gfCNCPoint2[3628] = {X 472.8698, Y 18.3782, Z -2.1667, A 0.000, B 0.000, C 0.000 }
gfCNCPoint2[3629] = {X 473.2481, Y 16.7251, Z -2.1667, A 0.000, B 0.000, C 0.000 }
gfCNCPoint2[3630] = {X 473.7840, Y 15.2312, Z -2.1667, A 0.000, B 0.000, C 0.000 }
gfCNCPoint2[3631] = {X 474.5174, Y 13.8238, Z -2.1667, A 0.000, B 0.000, C 0.000 }
gfCNCPoint2[3632] = {X 475.4350, Y 12.5288, Z -2.1667, A 0.000, B 0.000, C 0.000 }
gfCNCPoint2[3633] = {X 476.5196, Y 11.3702, Z -2.1667, A 0.000, B 0.000, C 0.000 }
gfCNCPoint2[3634] = {X 477.7513, Y 10.3694, Z -2.1667, A 0.000, B 0.000, C 0.000 }
gfCNCPoint2[3635] = {X 479.1074, Y 9.5448, Z -2.1667, A 0.000, B 0.000, C 0.000 }
gfCNCPoint2[3636] = {X 480.5628, Y 8.9117, Z -2.1667, A 0.000, B 0.000, C 0.000 }
gfCNCPoint2[3637] = {X 482.0905, Y 8.4819, Z -2.1667, A 0.000, B 0.000, C 0.000 }
gfCNCPoint2[3638] = {X 484.1725, Y 8.1580, Z -2.1667, A 0.000, B 0.000, C 0.000 }
gfCNCPoint2[3639] = {X 486.2764, Y 8.0437, Z -2.1667, A 0.000, B 0.000, C 0.000 }
gfCNCPoint2[3640] = {X 486.9693, Y 8.0316, Z -2.1667, A 0.000, B 0.000, C 0.000 }
gfCNCPoint2[3641] = {X 492.3824, Y 8.0316, Z -2.1667, A 0.000, B 0.000, C 0.000 }
gfCNCPoint2[3642] = {X 492.3824, Y 4.0316, Z -2.1667, A 0.000, B 0.000, C 0.000 }
gfCNCPoint2[3643] = {X 492.3824, Y 8.1116, Z -2.1667, A 0.000, B 0.000, C 0.000 }
gfCNCPoint2[3644] = {X 502.2056, Y 8.1116, Z -2.1667, A 0.000, B 0.000, C 0.000 }
gfCNCPoint2[3645] = {X 502.7355, Y 8.1157, Z -2.1667, A 0.000, B 0.000, C 0.000 }
gfCNCPoint2[3646] = {X 503.6347, Y 8.2236, Z -2.1667, A 0.000, B 0.000, C 0.000 }
gfCNCPoint2[3647] = {X 504.4878, Y 8.5280, Z -2.1667, A 0.000, B 0.000, C 0.000 }
gfCNCPoint2[3648] = {X 505.2522, Y 9.0137, Z -2.1667, A 0.000, B 0.000, C 0.000 }
gfCNCPoint2[3649] = {X 505.8902, Y 9.6567, Z -2.1667, A 0.000, B 0.000, C 0.000 }
gfCNCPoint2[3650] = {X 506.3699, Y 10.4249, Z -2.1667, A 0.000, B 0.000, C 0.000 }
gfCNCPoint2[3651] = {X 506.6676, Y 11.2803, Z -2.1667, A 0.000, B 0.000, C 0.000 }
gfCNCPoint2[3652] = {X 506.7685, Y 12.1804, Z -2.1667, A 0.000, B 0.000, C 0.000 }
gfCNCPoint2[3653] = {X 506.7685, Y 12.9781, Z -2.1667, A 0.000, B 0.000, C 0.000 }
gfCNCPoint2[3654] = {X 506.6667, Y 13.8835, Z -2.1667, A 0.000, B 0.000, C 0.000 }
gfCNCPoint2[3655] = {X 506.3666, Y 14.7437, Z -2.1667, A 0.000, B 0.000, C 0.000 }
gfCNCPoint2[3656] = {X 505.8831, Y 15.5159, Z -2.1667, A 0.000, B 0.000, C 0.000 }
gfCNCPoint2[3657] = {X 505.2403, Y 16.1615, Z -2.1667, A 0.000, B 0.000, C 0.000 }
gfCNCPoint2[3658] = {X 505.2402, Y 41.0273, Z -2.1667, A 0.000, B 0.000, C 0.000 }
gfCNCPoint2[3659] = {X 505.3177, Y 41.0889, Z -2.1667, A 0.000, B 0.000, C 0.000 }
gfCNCPoint2[3660] = {X 505.9239, Y 41.7232, Z -2.1667, A 0.000, B 0.000, C 0.000 }
gfCNCPoint2[3661] = {X 506.3805, Y 42.4724, Z -2.1667, A 0.000, B 0.000, C 0.000 }
gfCNCPoint2[3662] = {X 506.6664, Y 43.3019, Z -2.1667, A 0.000, B 0.000, C 0.000 }
gfCNCPoint2[3663] = {X 506.7683, Y 44.1734, Z -2.1667, A 0.000, B 0.000, C 0.000 }
gfCNCPoint2[3664] = {X 506.7685, Y 45.0000, Z -2.1667, A 0.000, B 0.000, C 0.000 }
gfCNCPoint2[3665] = {X 506.6662, Y 45.9079, Z -2.1667, A 0.000, B 0.000, C 0.000 }
gfCNCPoint2[3666] = {X 506.3644, Y 46.7702, Z -2.1667, A 0.000, B 0.000, C 0.000 }
gfCNCPoint2[3667] = {X 505.8784, Y 47.5438, Z -2.1667, A 0.000, B 0.000, C 0.000 }
gfCNCPoint2[3668] = {X 505.2323, Y 48.1899, Z -2.1667, A 0.000, B 0.000, C 0.000 }
gfCNCPoint2[3669] = {X 504.4587, Y 48.6760, Z -2.1667, A 0.000, B 0.000, C 0.000 }
gfCNCPoint2[3670] = {X 503.5964, Y 48.9777, Z -2.1667, A 0.000, B 0.000, C 0.000 }
gfCNCPoint2[3671] = {X 502.6885, Y 49.0800, Z -2.1667, A 0.000, B 0.000, C 0.000 }
gfCNCPoint2[3672] = {X 496.2450, Y 49.0800, Z -2.1667, A 0.000, B 0.000, C 0.000 }
gfCNCPoint2[3673] = {X 495.3416, Y 48.9787, Z -2.1667, A 0.000, B 0.000, C 0.000 }
gfCNCPoint2[3674] = {X 494.4831, Y 48.6799, Z -2.1667, A 0.000, B 0.000, C 0.000 }
gfCNCPoint2[3675] = {X 493.7120, Y 48.1985, Z -2.1667, A 0.000, B 0.000, C 0.000 }
gfCNCPoint2[3676] = {X 493.0667, Y 47.5582, Z -2.1667, A 0.000, B 0.000, C 0.000 }
gfCNCPoint2[3677] = {X 492.5791, Y 46.7909, Z -2.1667, A 0.000, B 0.000, C 0.000 }
gfCNCPoint2[3678] = {X 492.2736, Y 45.9348, Z -2.1667, A 0.000, B 0.000, C 0.000 }
gfCNCPoint2[3679] = {X 492.1652, Y 45.0322, Z -2.1667, A 0.000, B 0.000, C 0.000 }
gfCNCPoint2[3680] = {X 492.1654, Y 44.1527, Z -2.1667, A 0.000, B 0.000, C 0.000 }
gfCNCPoint2[3681] = {X 492.2760, Y 43.2637, Z -2.1667, A 0.000, B 0.000, C 0.000 }
gfCNCPoint2[3682] = {X 492.5779, Y 42.4203, Z -2.1667, A 0.000, B 0.000, C 0.000 }
gfCNCPoint2[3683] = {X 493.0566, Y 41.6631, Z -2.1667, A 0.000, B 0.000, C 0.000 }
gfCNCPoint2[3684] = {X 493.6890, Y 41.0287, Z -2.1667, A 0.000, B 0.000, C 0.000 }
gfCNCPoint2[3685] = {X 493.6890, Y 34.2338, Z -2.1667, A 0.000, B 0.000, C 0.000 }
gfCNCPoint2[3686] = {X 490.5769, Y 34.2338, Z -2.1667, A 0.000, B 0.000, C 0.000 }
gfCNCPoint2[3687] = {X 486.1773, Y 42.8013, Z -2.1667, A 0.000, B 0.000, C 0.000 }
gfCNCPoint2[3688] = {X 486.2188, Y 42.9100, Z -2.1667, A 0.000, B 0.000, C 0.000 }
gfCNCPoint2[3689] = {X 486.3746, Y 43.5327, Z -2.1667, A 0.000, B 0.000, C 0.000 }
gfCNCPoint2[3690] = {X 486.4309, Y 44.1720, Z -2.1667, A 0.000, B 0.000, C 0.000 }
gfCNCPoint2[3691] = {X 486.4310, Y 45.0000, Z -2.1667, A 0.000, B 0.000, C 0.000 }
gfCNCPoint2[3692] = {X 486.3287, Y 45.9079, Z -2.1667, A 0.000, B 0.000, C 0.000 }
gfCNCPoint2[3693] = {X 486.0270, Y 46.7702, Z -2.1667, A 0.000, B 0.000, C 0.000 }
gfCNCPoint2[3694] = {X 485.5409, Y 47.5438, Z -2.1667, A 0.000, B 0.000, C 0.000 }
gfCNCPoint2[3695] = {X 484.8949, Y 48.1899, Z -2.1667, A 0.000, B 0.000, C 0.000 }
gfCNCPoint2[3696] = {X 484.1213, Y 48.6760, Z -2.1667, A 0.000, B 0.000, C 0.000 }
gfCNCPoint2[3697] = {X 483.2589, Y 48.9777, Z -2.1667, A 0.000, B 0.000, C 0.000 }
gfCNCPoint2[3698] = {X 482.3510, Y 49.0800, Z -2.1667, A 0.000, B 0.000, C 0.000 }
gfCNCPoint2[3699] = {X 475.7650, Y 49.0800, Z -2.1667, A 0.000, B 0.000, C 0.000 }
gfCNCPoint2[3700] = {X 474.8571, Y 48.9777, Z -2.1667, A 0.000, B 0.000, C 0.000 }
gfCNCPoint2[3701] = {X 473.9947, Y 48.6760, Z -2.1667, A 0.000, B 0.000, C 0.000 }
gfCNCPoint2[3702] = {X 473.2211, Y 48.1899, Z -2.1667, A 0.000, B 0.000, C 0.000 }
gfCNCPoint2[3703] = {X 472.5751, Y 47.5438, Z -2.1667, A 0.000, B 0.000, C 0.000 }
gfCNCPoint2[3704] = {X 472.0890, Y 46.7702, Z -2.1667, A 0.000, B 0.000, C 0.000 }
gfCNCPoint2[3705] = {X 471.7873, Y 45.9079, Z -2.1667, A 0.000, B 0.000, C 0.000 }
gfCNCPoint2[3706] = {X 471.6850, Y 45.0000, Z -2.1667, A 0.000, B 0.000, C 0.000 }
gfCNCPoint2[3707] = {X 471.6853, Y 44.1527, Z -2.1667, A 0.000, B 0.000, C 0.000 }
gfCNCPoint2[3708] = {X 471.7809, Y 43.3294, Z -2.1667, A 0.000, B 0.000, C 0.000 }
gfCNCPoint2[3709] = {X 472.0408, Y 42.5424, Z -2.1667, A 0.000, B 0.000, C 0.000 }
gfCNCPoint2[3710] = {X 472.4544, Y 41.8242, Z -2.1667, A 0.000, B 0.000, C 0.000 }
gfCNCPoint2[3711] = {X 473.0046, Y 41.2044, Z -2.1667, A 0.000, B 0.000, C 0.000 }
gfCNCPoint2[3712] = {X 473.6687, Y 40.7085, Z -2.1667, A 0.000, B 0.000, C 0.000 }
gfCNCPoint2[3713] = {X 474.4193, Y 40.3571, Z -2.1667, A 0.000, B 0.000, C 0.000 }
gfCNCPoint2[3714] = {X 478.5504, Y 32.2709, Z -2.1667, A 0.000, B 0.000, C 0.000 }
gfCNCPoint2[3715] = {X 477.2669, Y 31.4235, Z -2.1667, A 0.000, B 0.000, C 0.000 }
gfCNCPoint2[3716] = {X 476.1112, Y 30.4087, Z -2.1667, A 0.000, B 0.000, C 0.000 }
gfCNCPoint2[3717] = {X 475.1050, Y 29.2455, Z -2.1667, A 0.000, B 0.000, C 0.000 }
gfCNCPoint2[3718] = {X 474.2671, Y 27.9557, Z -2.1667, A 0.000, B 0.000, C 0.000 }
gfCNCPoint2[3719] = {X 473.6133, Y 26.5636, Z -2.1667, A 0.000, B 0.000, C 0.000 }
gfCNCPoint2[3720] = {X 473.1559, Y 25.0952, Z -2.1667, A 0.000, B 0.000, C 0.000 }
gfCNCPoint2[3721] = {X 472.8464, Y 23.4362, Z -2.1667, A 0.000, B 0.000, C 0.000 }
gfCNCPoint2[3722] = {X 472.7080, Y 21.7543, Z -2.1667, A 0.000, B 0.000, C 0.000 }
gfCNCPoint2[3723] = {X 472.7422, Y 20.0670, Z -2.1667, A 0.000, B 0.000, C 0.000 }
gfCNCPoint2[3724] = {X 472.9486, Y 18.3920, Z -2.1667, A 0.000, B 0.000, C 0.000 }
gfCNCPoint2[3725] = {X 473.3251, Y 16.7469, Z -2.1667, A 0.000, B 0.000, C 0.000 }
gfCNCPoint2[3726] = {X 473.8573, Y 15.2633, Z -2.1667, A 0.000, B 0.000, C 0.000 }
gfCNCPoint2[3727] = {X 474.5857, Y 13.8655, Z -2.1667, A 0.000, B 0.000, C 0.000 }
gfCNCPoint2[3728] = {X 475.4969, Y 12.5794, Z -2.1667, A 0.000, B 0.000, C 0.000 }
gfCNCPoint2[3729] = {X 476.5742, Y 11.4287, Z -2.1667, A 0.000, B 0.000, C 0.000 }
gfCNCPoint2[3730] = {X 477.7975, Y 10.4348, Z -2.1667, A 0.000, B 0.000, C 0.000 }
gfCNCPoint2[3731] = {X 479.1442, Y 9.6158, Z -2.1667, A 0.000, B 0.000, C 0.000 }
gfCNCPoint2[3732] = {X 480.5896, Y 8.9871, Z -2.1667, A 0.000, B 0.000, C 0.000 }
gfCNCPoint2[3733] = {X 482.1069, Y 8.5602, Z -2.1667, A 0.000, B 0.000, C 0.000 }
gfCNCPoint2[3734] = {X 484.1812, Y 8.2375, Z -2.1667, A 0.000, B 0.000, C 0.000 }
gfCNCPoint2[3735] = {X 486.2773, Y 8.1237, Z -2.1667, A 0.000, B 0.000, C 0.000 }
gfCNCPoint2[3736] = {X 486.9700, Y 8.1116, Z -2.1667, A 0.000, B 0.000, C 0.000 }
gfCNCPoint2[3737] = {X 492.3824, Y 8.1116, Z -2.1667, A 0.000, B 0.000, C 0.000 }
gfCNCPoint2[3738] = {X 492.3824, Y 4.1116, Z -2.1667, A 0.000, B 0.000, C 0.000 }
gfCNCPoint2[3739] = {X 492.3824, Y 8.1916, Z -2.1667, A 0.000, B 0.000, C 0.000 }
gfCNCPoint2[3740] = {X 502.2053, Y 8.1916, Z -2.1667, A 0.000, B 0.000, C 0.000 }
gfCNCPoint2[3741] = {X 502.7348, Y 8.1957, Z -2.1667, A 0.000, B 0.000, C 0.000 }
gfCNCPoint2[3742] = {X 503.6164, Y 8.3015, Z -2.1667, A 0.000, B 0.000, C 0.000 }
gfCNCPoint2[3743] = {X 504.4526, Y 8.5999, Z -2.1667, A 0.000, B 0.000, C 0.000 }
gfCNCPoint2[3744] = {X 505.2021, Y 9.0761, Z -2.1667, A 0.000, B 0.000, C 0.000 }
gfCNCPoint2[3745] = {X 505.8274, Y 9.7063, Z -2.1667, A 0.000, B 0.000, C 0.000 }
gfCNCPoint2[3746] = {X 506.2977, Y 10.4594, Z -2.1667, A 0.000, B 0.000, C 0.000 }
gfCNCPoint2[3747] = {X 506.5896, Y 11.2980, Z -2.1667, A 0.000, B 0.000, C 0.000 }
gfCNCPoint2[3748] = {X 506.6885, Y 12.1804, Z -2.1667, A 0.000, B 0.000, C 0.000 }
gfCNCPoint2[3749] = {X 506.6883, Y 13.0192, Z -2.1667, A 0.000, B 0.000, C 0.000 }
gfCNCPoint2[3750] = {X 506.5796, Y 13.9051, Z -2.1667, A 0.000, B 0.000, C 0.000 }
gfCNCPoint2[3751] = {X 506.2772, Y 14.7448, Z -2.1667, A 0.000, B 0.000, C 0.000 }
gfCNCPoint2[3752] = {X 505.7961, Y 15.4965, Z -2.1667, A 0.000, B 0.000, C 0.000 }
gfCNCPoint2[3753] = {X 505.1603, Y 16.1229, Z -2.1667, A 0.000, B 0.000, C 0.000 }
gfCNCPoint2[3754] = {X 505.1602, Y 41.0659, Z -2.1667, A 0.000, B 0.000, C 0.000 }
gfCNCPoint2[3755] = {X 505.2992, Y 41.1782, Z -2.1667, A 0.000, B 0.000, C 0.000 }
gfCNCPoint2[3756] = {X 505.8855, Y 41.8047, Z -2.1667, A 0.000, B 0.000, C 0.000 }
gfCNCPoint2[3757] = {X 506.3246, Y 42.5419, Z -2.1667, A 0.000, B 0.000, C 0.000 }
gfCNCPoint2[3758] = {X 506.5965, Y 43.3558, Z -2.1667, A 0.000, B 0.000, C 0.000 }
gfCNCPoint2[3759] = {X 506.6885, Y 44.2089, Z -2.1667, A 0.000, B 0.000, C 0.000 }
gfCNCPoint2[3760] = {X 506.6885, Y 45.0000, Z -2.1667, A 0.000, B 0.000, C 0.000 }
gfCNCPoint2[3761] = {X 506.5882, Y 45.8901, Z -2.1667, A 0.000, B 0.000, C 0.000 }
gfCNCPoint2[3762] = {X 506.2924, Y 46.7355, Z -2.1667, A 0.000, B 0.000, C 0.000 }
gfCNCPoint2[3763] = {X 505.8158, Y 47.4940, Z -2.1667, A 0.000, B 0.000, C 0.000 }
gfCNCPoint2[3764] = {X 505.1825, Y 48.1273, Z -2.1667, A 0.000, B 0.000, C 0.000 }
gfCNCPoint2[3765] = {X 504.4240, Y 48.6039, Z -2.1667, A 0.000, B 0.000, C 0.000 }
gfCNCPoint2[3766] = {X 503.5786, Y 48.8997, Z -2.1667, A 0.000, B 0.000, C 0.000 }
gfCNCPoint2[3767] = {X 502.6885, Y 49.0000, Z -2.1667, A 0.000, B 0.000, C 0.000 }
gfCNCPoint2[3768] = {X 496.2450, Y 49.0000, Z -2.1667, A 0.000, B 0.000, C 0.000 }
gfCNCPoint2[3769] = {X 495.3549, Y 48.8997, Z -2.1667, A 0.000, B 0.000, C 0.000 }
gfCNCPoint2[3770] = {X 494.5095, Y 48.6039, Z -2.1667, A 0.000, B 0.000, C 0.000 }
gfCNCPoint2[3771] = {X 493.7510, Y 48.1273, Z -2.1667, A 0.000, B 0.000, C 0.000 }
gfCNCPoint2[3772] = {X 493.1177, Y 47.4939, Z -2.1667, A 0.000, B 0.000, C 0.000 }
gfCNCPoint2[3773] = {X 492.6411, Y 46.7355, Z -2.1667, A 0.000, B 0.000, C 0.000 }
gfCNCPoint2[3774] = {X 492.3453, Y 45.8900, Z -2.1667, A 0.000, B 0.000, C 0.000 }
gfCNCPoint2[3775] = {X 492.2450, Y 45.0000, Z -2.1667, A 0.000, B 0.000, C 0.000 }
gfCNCPoint2[3776] = {X 492.2454, Y 44.1538, Z -2.1667, A 0.000, B 0.000, C 0.000 }
gfCNCPoint2[3777] = {X 492.3560, Y 43.2730, Z -2.1667, A 0.000, B 0.000, C 0.000 }
gfCNCPoint2[3778] = {X 492.6582, Y 42.4382, Z -2.1667, A 0.000, B 0.000, C 0.000 }
gfCNCPoint2[3779] = {X 493.1371, Y 41.6907, Z -2.1667, A 0.000, B 0.000, C 0.000 }
gfCNCPoint2[3780] = {X 493.7690, Y 41.0672, Z -2.1667, A 0.000, B 0.000, C 0.000 }
gfCNCPoint2[3781] = {X 493.7690, Y 34.1538, Z -2.1667, A 0.000, B 0.000, C 0.000 }
gfCNCPoint2[3782] = {X 490.7723, Y 34.1538, Z -2.1667, A 0.000, B 0.000, C 0.000 }
gfCNCPoint2[3783] = {X 490.5297, Y 34.1507, Z -2.1667, A 0.000, B 0.000, C 0.000 }
gfCNCPoint2[3784] = {X 486.0898, Y 42.7965, Z -2.1667, A 0.000, B 0.000, C 0.000 }
gfCNCPoint2[3785] = {X 486.1470, Y 42.9477, Z -2.1667, A 0.000, B 0.000, C 0.000 }
gfCNCPoint2[3786] = {X 486.2997, Y 43.5701, Z -2.1667, A 0.000, B 0.000, C 0.000 }
gfCNCPoint2[3787] = {X 486.3510, Y 44.2089, Z -2.1667, A 0.000, B 0.000, C 0.000 }
gfCNCPoint2[3788] = {X 486.3510, Y 45.0000, Z -2.1667, A 0.000, B 0.000, C 0.000 }
gfCNCPoint2[3789] = {X 486.2507, Y 45.8901, Z -2.1667, A 0.000, B 0.000, C 0.000 }
gfCNCPoint2[3790] = {X 485.9549, Y 46.7355, Z -2.1667, A 0.000, B 0.000, C 0.000 }
gfCNCPoint2[3791] = {X 485.4783, Y 47.4940, Z -2.1667, A 0.000, B 0.000, C 0.000 }
gfCNCPoint2[3792] = {X 484.8450, Y 48.1273, Z -2.1667, A 0.000, B 0.000, C 0.000 }
gfCNCPoint2[3793] = {X 484.0866, Y 48.6039, Z -2.1667, A 0.000, B 0.000, C 0.000 }
gfCNCPoint2[3794] = {X 483.2411, Y 48.8997, Z -2.1667, A 0.000, B 0.000, C 0.000 }
gfCNCPoint2[3795] = {X 482.3510, Y 49.0000, Z -2.1667, A 0.000, B 0.000, C 0.000 }
gfCNCPoint2[3796] = {X 475.7650, Y 49.0000, Z -2.1667, A 0.000, B 0.000, C 0.000 }
gfCNCPoint2[3797] = {X 474.8749, Y 48.8997, Z -2.1667, A 0.000, B 0.000, C 0.000 }
gfCNCPoint2[3798] = {X 474.0294, Y 48.6039, Z -2.1667, A 0.000, B 0.000, C 0.000 }
gfCNCPoint2[3799] = {X 473.2710, Y 48.1273, Z -2.1667, A 0.000, B 0.000, C 0.000 }
gfCNCPoint2[3800] = {X 472.6376, Y 47.4940, Z -2.1667, A 0.000, B 0.000, C 0.000 }
gfCNCPoint2[3801] = {X 472.1611, Y 46.7355, Z -2.1667, A 0.000, B 0.000, C 0.000 }
gfCNCPoint2[3802] = {X 471.8652, Y 45.8901, Z -2.1667, A 0.000, B 0.000, C 0.000 }
gfCNCPoint2[3803] = {X 471.7650, Y 45.0000, Z -2.1667, A 0.000, B 0.000, C 0.000 }
gfCNCPoint2[3804] = {X 471.7653, Y 44.1538, Z -2.1667, A 0.000, B 0.000, C 0.000 }
gfCNCPoint2[3805] = {X 471.8601, Y 43.3414, Z -2.1667, A 0.000, B 0.000, C 0.000 }
gfCNCPoint2[3806] = {X 472.1182, Y 42.5654, Z -2.1667, A 0.000, B 0.000, C 0.000 }
gfCNCPoint2[3807] = {X 472.5286, Y 41.8580, Z -2.1667, A 0.000, B 0.000, C 0.000 }
gfCNCPoint2[3808] = {X 473.0744, Y 41.2489, Z -2.1667, A 0.000, B 0.000, C 0.000 }
gfCNCPoint2[3809] = {X 473.7327, Y 40.7635, Z -2.1667, A 0.000, B 0.000, C 0.000 }
gfCNCPoint2[3810] = {X 474.4759, Y 40.4222, Z -2.1667, A 0.000, B 0.000, C 0.000 }
gfCNCPoint2[3811] = {X 478.6566, Y 32.2388, Z -2.1667, A 0.000, B 0.000, C 0.000 }
gfCNCPoint2[3812] = {X 477.3663, Y 31.3985, Z -2.1667, A 0.000, B 0.000, C 0.000 }
gfCNCPoint2[3813] = {X 476.2040, Y 30.3885, Z -2.1667, A 0.000, B 0.000, C 0.000 }
gfCNCPoint2[3814] = {X 475.1919, Y 29.2280, Z -2.1667, A 0.000, B 0.000, C 0.000 }
gfCNCPoint2[3815] = {X 474.3494, Y 27.9391, Z -2.1667, A 0.000, B 0.000, C 0.000 }
gfCNCPoint2[3816] = {X 473.6925, Y 26.5464, Z -2.1667, A 0.000, B 0.000, C 0.000 }
gfCNCPoint2[3817] = {X 473.2337, Y 25.0766, Z -2.1667, A 0.000, B 0.000, C 0.000 }
gfCNCPoint2[3818] = {X 472.9257, Y 23.4256, Z -2.1667, A 0.000, B 0.000, C 0.000 }
gfCNCPoint2[3819] = {X 472.7880, Y 21.7518, Z -2.1667, A 0.000, B 0.000, C 0.000 }
gfCNCPoint2[3820] = {X 472.8220, Y 20.0727, Z -2.1667, A 0.000, B 0.000, C 0.000 }
gfCNCPoint2[3821] = {X 473.0274, Y 18.4059, Z -2.1667, A 0.000, B 0.000, C 0.000 }
gfCNCPoint2[3822] = {X 473.4020, Y 16.7687, Z -2.1667, A 0.000, B 0.000, C 0.000 }
gfCNCPoint2[3823] = {X 473.9306, Y 15.2953, Z -2.1667, A 0.000, B 0.000, C 0.000 }
gfCNCPoint2[3824] = {X 474.6540, Y 13.9072, Z -2.1667, A 0.000, B 0.000, C 0.000 }
gfCNCPoint2[3825] = {X 475.5589, Y 12.6300, Z -2.1667, A 0.000, B 0.000, C 0.000 }
gfCNCPoint2[3826] = {X 476.6287, Y 11.4872, Z -2.1667, A 0.000, B 0.000, C 0.000 }
gfCNCPoint2[3827] = {X 477.8436, Y 10.5001, Z -2.1667, A 0.000, B 0.000, C 0.000 }
gfCNCPoint2[3828] = {X 479.1811, Y 9.6869, Z -2.1667, A 0.000, B 0.000, C 0.000 }
gfCNCPoint2[3829] = {X 480.6165, Y 9.0625, Z -2.1667, A 0.000, B 0.000, C 0.000 }
gfCNCPoint2[3830] = {X 482.1233, Y 8.6385, Z -2.1667, A 0.000, B 0.000, C 0.000 }
gfCNCPoint2[3831] = {X 484.1898, Y 8.3170, Z -2.1667, A 0.000, B 0.000, C 0.000 }
gfCNCPoint2[3832] = {X 486.2782, Y 8.2037, Z -2.1667, A 0.000, B 0.000, C 0.000 }
gfCNCPoint2[3833] = {X 486.9707, Y 8.1916, Z -2.1667, A 0.000, B 0.000, C 0.000 }
gfCNCPoint2[3834] = {X 492.3824, Y 8.1916, Z -2.1667, A 0.000, B 0.000, C 0.000 }
gfCNCPoint2[3835] = {X 492.3824, Y 4.1116, Z -2.1667, A 0.000, B 0.000, C 0.000 }
gfCNCPoint2[3836] = {X 492.3824, Y 4.1116, Z 0.8333, A 0.000, B 0.000, C 0.000 }
gfCNCPoint2[3837] = {X 492.3824, Y 4.1116, Z 11.0000, A 0.000, B 0.000, C 0.000 }
gfCNCPoint2[3838] = {X 533.9641, Y 3.7913, Z 11.0000, A 0.000, B 0.000, C 0.000 }
gfCNCPoint2[3839] = {X 533.9641, Y 3.7913, Z 0.8333, A 0.000, B 0.000, C 0.000 }
gfCNCPoint2[3840] = {X 533.9641, Y 3.7913, Z -2.1667, A 0.000, B 0.000, C 0.000 }
gfCNCPoint2[3841] = {X 533.9640, Y 7.8713, Z -2.1667, A 0.000, B 0.000, C 0.000 }
gfCNCPoint2[3842] = {X 543.7499, Y 7.8716, Z -2.1667, A 0.000, B 0.000, C 0.000 }
gfCNCPoint2[3843] = {X 544.7300, Y 7.9571, Z -2.1667, A 0.000, B 0.000, C 0.000 }
gfCNCPoint2[3844] = {X 545.6654, Y 8.2619, Z -2.1667, A 0.000, B 0.000, C 0.000 }
gfCNCPoint2[3845] = {X 546.5077, Y 8.7702, Z -2.1667, A 0.000, B 0.000, C 0.000 }
gfCNCPoint2[3846] = {X 547.2133, Y 9.4557, Z -2.1667, A 0.000, B 0.000, C 0.000 }
gfCNCPoint2[3847] = {X 547.7458, Y 10.2829, Z -2.1667, A 0.000, B 0.000, C 0.000 }
gfCNCPoint2[3848] = {X 548.0776, Y 11.2091, Z -2.1667, A 0.000, B 0.000, C 0.000 }
gfCNCPoint2[3849] = {X 548.1914, Y 12.1862, Z -2.1667, A 0.000, B 0.000, C 0.000 }
gfCNCPoint2[3850] = {X 548.1912, Y 13.0225, Z -2.1667, A 0.000, B 0.000, C 0.000 }
gfCNCPoint2[3851] = {X 548.0827, Y 13.9408, Z -2.1667, A 0.000, B 0.000, C 0.000 }
gfCNCPoint2[3852] = {X 547.7812, Y 14.8150, Z -2.1667, A 0.000, B 0.000, C 0.000 }
gfCNCPoint2[3853] = {X 547.3006, Y 15.6050, Z -2.1667, A 0.000, B 0.000, C 0.000 }
gfCNCPoint2[3854] = {X 546.6629, Y 16.2746, Z -2.1667, A 0.000, B 0.000, C 0.000 }
gfCNCPoint2[3855] = {X 546.6631, Y 40.9131, Z -2.1667, A 0.000, B 0.000, C 0.000 }
gfCNCPoint2[3856] = {X 546.6855, Y 40.9311, Z -2.1667, A 0.000, B 0.000, C 0.000 }
gfCNCPoint2[3857] = {X 547.3155, Y 41.6010, Z -2.1667, A 0.000, B 0.000, C 0.000 }
gfCNCPoint2[3858] = {X 547.7895, Y 42.3891, Z -2.1667, A 0.000, B 0.000, C 0.000 }
gfCNCPoint2[3859] = {X 548.0859, Y 43.2597, Z -2.1667, A 0.000, B 0.000, C 0.000 }
gfCNCPoint2[3860] = {X 548.1913, Y 44.1733, Z -2.1667, A 0.000, B 0.000, C 0.000 }
gfCNCPoint2[3861] = {X 548.1914, Y 45.0006, Z -2.1667, A 0.000, B 0.000, C 0.000 }
gfCNCPoint2[3862] = {X 548.0776, Y 45.9777, Z -2.1667, A 0.000, B 0.000, C 0.000 }
gfCNCPoint2[3863] = {X 547.7458, Y 46.9039, Z -2.1667, A 0.000, B 0.000, C 0.000 }
gfCNCPoint2[3864] = {X 547.2133, Y 47.7311, Z -2.1667, A 0.000, B 0.000, C 0.000 }
gfCNCPoint2[3865] = {X 546.5077, Y 48.4165, Z -2.1667, A 0.000, B 0.000, C 0.000 }
gfCNCPoint2[3866] = {X 545.6653, Y 48.9248, Z -2.1667, A 0.000, B 0.000, C 0.000 }
gfCNCPoint2[3867] = {X 544.7300, Y 49.2295, Z -2.1667, A 0.000, B 0.000, C 0.000 }
gfCNCPoint2[3868] = {X 543.7499, Y 49.3149, Z -2.1667, A 0.000, B 0.000, C 0.000 }
gfCNCPoint2[3869] = {X 524.0447, Y 49.3155, Z -2.1667, A 0.000, B 0.000, C 0.000 }
gfCNCPoint2[3870] = {X 523.4982, Y 49.9494, Z -2.1667, A 0.000, B 0.000, C 0.000 }
gfCNCPoint2[3871] = {X 522.8433, Y 50.4706, Z -2.1667, A 0.000, B 0.000, C 0.000 }
gfCNCPoint2[3872] = {X 522.1029, Y 50.8609, Z -2.1667, A 0.000, B 0.000, C 0.000 }
gfCNCPoint2[3873] = {X 521.3028, Y 51.1066, Z -2.1667, A 0.000, B 0.000, C 0.000 }
gfCNCPoint2[3874] = {X 520.4709, Y 51.1991, Z -2.1667, A 0.000, B 0.000, C 0.000 }
gfCNCPoint2[3875] = {X 519.7998, Y 51.1991, Z -2.1667, A 0.000, B 0.000, C 0.000 }
gfCNCPoint2[3876] = {X 518.8385, Y 51.0908, Z -2.1667, A 0.000, B 0.000, C 0.000 }
gfCNCPoint2[3877] = {X 517.9254, Y 50.7713, Z -2.1667, A 0.000, B 0.000, C 0.000 }
gfCNCPoint2[3878] = {X 517.1063, Y 50.2566, Z -2.1667, A 0.000, B 0.000, C 0.000 }
gfCNCPoint2[3879] = {X 516.4223, Y 49.5726, Z -2.1667, A 0.000, B 0.000, C 0.000 }
gfCNCPoint2[3880] = {X 515.9076, Y 48.7535, Z -2.1667, A 0.000, B 0.000, C 0.000 }
gfCNCPoint2[3881] = {X 515.5881, Y 47.8404, Z -2.1667, A 0.000, B 0.000, C 0.000 }
gfCNCPoint2[3882] = {X 515.4798, Y 46.8791, Z -2.1667, A 0.000, B 0.000, C 0.000 }
gfCNCPoint2[3883] = {X 515.4798, Y 39.9011, Z -2.1667, A 0.000, B 0.000, C 0.000 }
gfCNCPoint2[3884] = {X 515.5869, Y 38.9451, Z -2.1667, A 0.000, B 0.000, C 0.000 }
gfCNCPoint2[3885] = {X 515.9029, Y 38.0365, Z -2.1667, A 0.000, B 0.000, C 0.000 }
gfCNCPoint2[3886] = {X 516.4121, Y 37.2204, Z -2.1667, A 0.000, B 0.000, C 0.000 }
gfCNCPoint2[3887] = {X 517.0893, Y 36.5372, Z -2.1667, A 0.000, B 0.000, C 0.000 }
gfCNCPoint2[3888] = {X 517.9010, Y 36.0208, Z -2.1667, A 0.000, B 0.000, C 0.000 }
gfCNCPoint2[3889] = {X 518.8067, Y 35.6968, Z -2.1667, A 0.000, B 0.000, C 0.000 }
gfCNCPoint2[3890] = {X 519.7617, Y 35.5813, Z -2.1667, A 0.000, B 0.000, C 0.000 }
gfCNCPoint2[3891] = {X 520.5269, Y 35.5815, Z -2.1667, A 0.000, B 0.000, C 0.000 }
gfCNCPoint2[3892] = {X 521.3535, Y 35.6728, Z -2.1667, A 0.000, B 0.000, C 0.000 }
gfCNCPoint2[3893] = {X 522.1474, Y 35.9208, Z -2.1667, A 0.000, B 0.000, C 0.000 }
gfCNCPoint2[3894] = {X 522.8790, Y 36.3164, Z -2.1667, A 0.000, B 0.000, C 0.000 }
gfCNCPoint2[3895] = {X 523.5213, Y 36.8448, Z -2.1667, A 0.000, B 0.000, C 0.000 }
gfCNCPoint2[3896] = {X 524.0504, Y 37.4865, Z -2.1667, A 0.000, B 0.000, C 0.000 }
gfCNCPoint2[3897] = {X 534.6319, Y 37.4871, Z -2.1667, A 0.000, B 0.000, C 0.000 }
gfCNCPoint2[3898] = {X 534.6319, Y 33.9648, Z -2.1667, A 0.000, B 0.000, C 0.000 }
gfCNCPoint2[3899] = {X 530.1092, Y 33.9661, Z -2.1667, A 0.000, B 0.000, C 0.000 }
gfCNCPoint2[3900] = {X 529.5770, Y 34.6102, Z -2.1667, A 0.000, B 0.000, C 0.000 }
gfCNCPoint2[3901] = {X 528.9308, Y 35.1398, Z -2.1667, A 0.000, B 0.000, C 0.000 }
gfCNCPoint2[3902] = {X 528.1947, Y 35.5352, Z -2.1667, A 0.000, B 0.000, C 0.000 }
gfCNCPoint2[3903] = {X 527.3963, Y 35.7814, Z -2.1667, A 0.000, B 0.000, C 0.000 }
gfCNCPoint2[3904] = {X 526.5655, Y 35.8693, Z -2.1667, A 0.000, B 0.000, C 0.000 }
gfCNCPoint2[3905] = {X 525.8868, Y 35.8694, Z -2.1667, A 0.000, B 0.000, C 0.000 }
gfCNCPoint2[3906] = {X 524.9255, Y 35.7611, Z -2.1667, A 0.000, B 0.000, C 0.000 }
gfCNCPoint2[3907] = {X 524.0124, Y 35.4416, Z -2.1667, A 0.000, B 0.000, C 0.000 }
gfCNCPoint2[3908] = {X 523.1933, Y 34.9270, Z -2.1667, A 0.000, B 0.000, C 0.000 }
gfCNCPoint2[3909] = {X 522.5092, Y 34.2429, Z -2.1667, A 0.000, B 0.000, C 0.000 }
gfCNCPoint2[3910] = {X 521.9946, Y 33.4238, Z -2.1667, A 0.000, B 0.000, C 0.000 }
gfCNCPoint2[3911] = {X 521.6751, Y 32.5107, Z -2.1667, A 0.000, B 0.000, C 0.000 }
gfCNCPoint2[3912] = {X 521.5668, Y 31.5495, Z -2.1667, A 0.000, B 0.000, C 0.000 }
gfCNCPoint2[3913] = {X 521.5668, Y 24.5714, Z -2.1667, A 0.000, B 0.000, C 0.000 }
gfCNCPoint2[3914] = {X 521.6739, Y 23.6153, Z -2.1667, A 0.000, B 0.000, C 0.000 }
gfCNCPoint2[3915] = {X 521.9900, Y 22.7066, Z -2.1667, A 0.000, B 0.000, C 0.000 }
gfCNCPoint2[3916] = {X 522.4994, Y 21.8904, Z -2.1667, A 0.000, B 0.000, C 0.000 }
gfCNCPoint2[3917] = {X 523.1768, Y 21.2071, Z -2.1667, A 0.000, B 0.000, C 0.000 }
gfCNCPoint2[3918] = {X 523.9886, Y 20.6908, Z -2.1667, A 0.000, B 0.000, C 0.000 }
gfCNCPoint2[3919] = {X 524.8946, Y 20.3669, Z -2.1667, A 0.000, B 0.000, C 0.000 }
gfCNCPoint2[3920] = {X 525.8498, Y 20.2516, Z -2.1667, A 0.000, B 0.000, C 0.000 }
gfCNCPoint2[3921] = {X 526.5695, Y 20.2516, Z -2.1667, A 0.000, B 0.000, C 0.000 }
gfCNCPoint2[3922] = {X 527.3947, Y 20.3392, Z -2.1667, A 0.000, B 0.000, C 0.000 }
gfCNCPoint2[3923] = {X 528.1880, Y 20.5829, Z -2.1667, A 0.000, B 0.000, C 0.000 }
gfCNCPoint2[3924] = {X 528.9201, Y 20.9739, Z -2.1667, A 0.000, B 0.000, C 0.000 }
gfCNCPoint2[3925] = {X 529.5638, Y 21.4976, Z -2.1667, A 0.000, B 0.000, C 0.000 }
gfCNCPoint2[3926] = {X 530.0956, Y 22.1347, Z -2.1667, A 0.000, B 0.000, C 0.000 }
gfCNCPoint2[3927] = {X 534.6319, Y 22.1350, Z -2.1667, A 0.000, B 0.000, C 0.000 }
gfCNCPoint2[3928] = {X 534.6319, Y 19.7012, Z -2.1667, A 0.000, B 0.000, C 0.000 }
gfCNCPoint2[3929] = {X 524.1927, Y 19.7007, Z -2.1667, A 0.000, B 0.000, C 0.000 }
gfCNCPoint2[3930] = {X 523.6603, Y 20.3456, Z -2.1667, A 0.000, B 0.000, C 0.000 }
gfCNCPoint2[3931] = {X 523.0136, Y 20.8758, Z -2.1667, A 0.000, B 0.000, C 0.000 }
gfCNCPoint2[3932] = {X 522.2768, Y 21.2715, Z -2.1667, A 0.000, B 0.000, C 0.000 }
gfCNCPoint2[3933] = {X 521.4776, Y 21.5178, Z -2.1667, A 0.000, B 0.000, C 0.000 }
gfCNCPoint2[3934] = {X 520.6460, Y 21.6056, Z -2.1667, A 0.000, B 0.000, C 0.000 }
gfCNCPoint2[3935] = {X 519.9691, Y 21.6057, Z -2.1667, A 0.000, B 0.000, C 0.000 }
gfCNCPoint2[3936] = {X 519.0078, Y 21.4974, Z -2.1667, A 0.000, B 0.000, C 0.000 }
gfCNCPoint2[3937] = {X 518.0947, Y 21.1779, Z -2.1667, A 0.000, B 0.000, C 0.000 }
gfCNCPoint2[3938] = {X 517.2756, Y 20.6632, Z -2.1667, A 0.000, B 0.000, C 0.000 }
gfCNCPoint2[3939] = {X 516.5916, Y 19.9792, Z -2.1667, A 0.000, B 0.000, C 0.000 }
gfCNCPoint2[3940] = {X 516.0769, Y 19.1601, Z -2.1667, A 0.000, B 0.000, C 0.000 }
gfCNCPoint2[3941] = {X 515.7574, Y 18.2470, Z -2.1667, A 0.000, B 0.000, C 0.000 }
gfCNCPoint2[3942] = {X 515.6491, Y 17.2857, Z -2.1667, A 0.000, B 0.000, C 0.000 }
gfCNCPoint2[3943] = {X 515.6491, Y 10.3077, Z -2.1667, A 0.000, B 0.000, C 0.000 }
gfCNCPoint2[3944] = {X 515.7562, Y 9.3519, Z -2.1667, A 0.000, B 0.000, C 0.000 }
gfCNCPoint2[3945] = {X 516.0720, Y 8.4435, Z -2.1667, A 0.000, B 0.000, C 0.000 }
gfCNCPoint2[3946] = {X 516.5811, Y 7.6275, Z -2.1667, A 0.000, B 0.000, C 0.000 }
gfCNCPoint2[3947] = {X 517.2580, Y 6.9443, Z -2.1667, A 0.000, B 0.000, C 0.000 }
gfCNCPoint2[3948] = {X 518.0693, Y 6.4278, Z -2.1667, A 0.000, B 0.000, C 0.000 }
gfCNCPoint2[3949] = {X 518.9748, Y 6.1037, Z -2.1667, A 0.000, B 0.000, C 0.000 }
gfCNCPoint2[3950] = {X 519.9296, Y 5.9879, Z -2.1667, A 0.000, B 0.000, C 0.000 }
gfCNCPoint2[3951] = {X 520.6502, Y 5.9879, Z -2.1667, A 0.000, B 0.000, C 0.000 }
gfCNCPoint2[3952] = {X 521.4758, Y 6.0752, Z -2.1667, A 0.000, B 0.000, C 0.000 }
gfCNCPoint2[3953] = {X 522.2695, Y 6.3188, Z -2.1667, A 0.000, B 0.000, C 0.000 }
gfCNCPoint2[3954] = {X 523.0019, Y 6.7098, Z -2.1667, A 0.000, B 0.000, C 0.000 }
gfCNCPoint2[3955] = {X 523.6460, Y 7.2336, Z -2.1667, A 0.000, B 0.000, C 0.000 }
gfCNCPoint2[3956] = {X 524.1780, Y 7.8710, Z -2.1667, A 0.000, B 0.000, C 0.000 }
gfCNCPoint2[3957] = {X 533.9640, Y 7.8713, Z -2.1667, A 0.000, B 0.000, C 0.000 }
gfCNCPoint2[3958] = {X 533.9641, Y 3.8713, Z -2.1667, A 0.000, B 0.000, C 0.000 }
gfCNCPoint2[3959] = {X 533.9640, Y 7.9513, Z -2.1667, A 0.000, B 0.000, C 0.000 }
gfCNCPoint2[3960] = {X 543.7510, Y 7.9516, Z -2.1667, A 0.000, B 0.000, C 0.000 }
gfCNCPoint2[3961] = {X 544.7131, Y 8.0353, Z -2.1667, A 0.000, B 0.000, C 0.000 }
gfCNCPoint2[3962] = {X 545.6314, Y 8.3343, Z -2.1667, A 0.000, B 0.000, C 0.000 }
gfCNCPoint2[3963] = {X 546.4583, Y 8.8331, Z -2.1667, A 0.000, B 0.000, C 0.000 }
gfCNCPoint2[3964] = {X 547.1511, Y 9.5060, Z -2.1667, A 0.000, B 0.000, C 0.000 }
gfCNCPoint2[3965] = {X 547.6739, Y 10.3180, Z -2.1667, A 0.000, B 0.000, C 0.000 }
gfCNCPoint2[3966] = {X 547.9996, Y 11.2271, Z -2.1667, A 0.000, B 0.000, C 0.000 }
gfCNCPoint2[3967] = {X 548.1114, Y 12.1864, Z -2.1667, A 0.000, B 0.000, C 0.000 }
gfCNCPoint2[3968] = {X 548.1112, Y 13.0217, Z -2.1667, A 0.000, B 0.000, C 0.000 }
gfCNCPoint2[3969] = {X 548.0026, Y 13.9320, Z -2.1667, A 0.000, B 0.000, C 0.000 }
gfCNCPoint2[3970] = {X 547.7009, Y 14.7977, Z -2.1667, A 0.000, B 0.000, C 0.000 }
gfCNCPoint2[3971] = {X 547.2202, Y 15.5783, Z -2.1667, A 0.000, B 0.000, C 0.000 }
gfCNCPoint2[3972] = {X 546.5829, Y 16.2373, Z -2.1667, A 0.000, B 0.000, C 0.000 }
gfCNCPoint2[3973] = {X 546.5831, Y 40.9514, Z -2.1667, A 0.000, B 0.000, C 0.000 }
gfCNCPoint2[3974] = {X 546.6343, Y 40.9926, Z -2.1667, A 0.000, B 0.000, C 0.000 }
gfCNCPoint2[3975] = {X 547.2523, Y 41.6500, Z -2.1667, A 0.000, B 0.000, C 0.000 }
gfCNCPoint2[3976] = {X 547.7172, Y 42.4234, Z -2.1667, A 0.000, B 0.000, C 0.000 }
gfCNCPoint2[3977] = {X 548.0079, Y 43.2776, Z -2.1667, A 0.000, B 0.000, C 0.000 }
gfCNCPoint2[3978] = {X 548.1113, Y 44.1740, Z -2.1667, A 0.000, B 0.000, C 0.000 }
gfCNCPoint2[3979] = {X 548.1114, Y 45.0004, Z -2.1667, A 0.000, B 0.000, C 0.000 }
gfCNCPoint2[3980] = {X 547.9996, Y 45.9597, Z -2.1667, A 0.000, B 0.000, C 0.000 }
gfCNCPoint2[3981] = {X 547.6739, Y 46.8688, Z -2.1667, A 0.000, B 0.000, C 0.000 }
gfCNCPoint2[3982] = {X 547.1511, Y 47.6808, Z -2.1667, A 0.000, B 0.000, C 0.000 }
gfCNCPoint2[3983] = {X 546.4583, Y 48.3535, Z -2.1667, A 0.000, B 0.000, C 0.000 }
gfCNCPoint2[3984] = {X 545.6314, Y 48.8523, Z -2.1667, A 0.000, B 0.000, C 0.000 }
gfCNCPoint2[3985] = {X 544.7131, Y 49.1513, Z -2.1667, A 0.000, B 0.000, C 0.000 }
gfCNCPoint2[3986] = {X 543.7510, Y 49.2349, Z -2.1667, A 0.000, B 0.000, C 0.000 }
gfCNCPoint2[3987] = {X 524.0032, Y 49.2355, Z -2.1667, A 0.000, B 0.000, C 0.000 }
gfCNCPoint2[3988] = {X 523.4665, Y 49.8688, Z -2.1667, A 0.000, B 0.000, C 0.000 }
gfCNCPoint2[3989] = {X 522.8204, Y 50.3899, Z -2.1667, A 0.000, B 0.000, C 0.000 }
gfCNCPoint2[3990] = {X 522.0879, Y 50.7805, Z -2.1667, A 0.000, B 0.000, C 0.000 }
gfCNCPoint2[3991] = {X 521.2951, Y 51.0265, Z -2.1667, A 0.000, B 0.000, C 0.000 }
gfCNCPoint2[3992] = {X 520.4702, Y 51.1191, Z -2.1667, A 0.000, B 0.000, C 0.000 }
gfCNCPoint2[3993] = {X 519.7998, Y 51.1191, Z -2.1667, A 0.000, B 0.000, C 0.000 }
gfCNCPoint2[3994] = {X 518.8563, Y 51.0128, Z -2.1667, A 0.000, B 0.000, C 0.000 }
gfCNCPoint2[3995] = {X 517.9601, Y 50.6992, Z -2.1667, A 0.000, B 0.000, C 0.000 }
gfCNCPoint2[3996] = {X 517.1562, Y 50.1941, Z -2.1667, A 0.000, B 0.000, C 0.000 }
gfCNCPoint2[3997] = {X 516.4848, Y 49.5227, Z -2.1667, A 0.000, B 0.000, C 0.000 }
gfCNCPoint2[3998] = {X 515.9797, Y 48.7188, Z -2.1667, A 0.000, B 0.000, C 0.000 }
gfCNCPoint2[3999] = {X 515.6661, Y 47.8226, Z -2.1667, A 0.000, B 0.000, C 0.000 }
gfCNCPoint2[4000] = {X 515.5598, Y 46.8791, Z -2.1667, A 0.000, B 0.000, C 0.000 }
gfCNCPoint2[4001] = {X 515.5598, Y 39.9011, Z -2.1667, A 0.000, B 0.000, C 0.000 }
gfCNCPoint2[4002] = {X 515.6649, Y 38.9628, Z -2.1667, A 0.000, B 0.000, C 0.000 }
gfCNCPoint2[4003] = {X 515.9751, Y 38.0710, Z -2.1667, A 0.000, B 0.000, C 0.000 }
gfCNCPoint2[4004] = {X 516.4749, Y 37.2700, Z -2.1667, A 0.000, B 0.000, C 0.000 }
gfCNCPoint2[4005] = {X 517.1395, Y 36.5995, Z -2.1667, A 0.000, B 0.000, C 0.000 }
gfCNCPoint2[4006] = {X 517.9361, Y 36.0926, Z -2.1667, A 0.000, B 0.000, C 0.000 }
gfCNCPoint2[4007] = {X 518.8251, Y 35.7746, Z -2.1667, A 0.000, B 0.000, C 0.000 }
gfCNCPoint2[4008] = {X 519.7624, Y 35.6613, Z -2.1667, A 0.000, B 0.000, C 0.000 }
gfCNCPoint2[4009] = {X 520.5258, Y 35.6615, Z -2.1667, A 0.000, B 0.000, C 0.000 }
gfCNCPoint2[4010] = {X 521.3455, Y 35.7528, Z -2.1667, A 0.000, B 0.000, C 0.000 }
gfCNCPoint2[4011] = {X 522.1319, Y 36.0012, Z -2.1667, A 0.000, B 0.000, C 0.000 }
gfCNCPoint2[4012] = {X 522.8554, Y 36.3970, Z -2.1667, A 0.000, B 0.000, C 0.000 }
gfCNCPoint2[4013] = {X 523.4886, Y 36.9255, Z -2.1667, A 0.000, B 0.000, C 0.000 }
gfCNCPoint2[4014] = {X 524.0076, Y 37.5665, Z -2.1667, A 0.000, B 0.000, C 0.000 }
gfCNCPoint2[4015] = {X 534.7119, Y 37.5671, Z -2.1667, A 0.000, B 0.000, C 0.000 }
gfCNCPoint2[4016] = {X 534.7119, Y 33.8848, Z -2.1667, A 0.000, B 0.000, C 0.000 }
gfCNCPoint2[4017] = {X 530.0660, Y 33.8842, Z -2.1667, A 0.000, B 0.000, C 0.000 }
gfCNCPoint2[4018] = {X 530.0421, Y 33.9226, Z -2.1667, A 0.000, B 0.000, C 0.000 }
gfCNCPoint2[4019] = {X 529.5198, Y 34.5544, Z -2.1667, A 0.000, B 0.000, C 0.000 }
gfCNCPoint2[4020] = {X 528.8856, Y 35.0738, Z -2.1667, A 0.000, B 0.000, C 0.000 }
gfCNCPoint2[4021] = {X 528.1634, Y 35.4616, Z -2.1667, A 0.000, B 0.000, C 0.000 }
gfCNCPoint2[4022] = {X 527.3800, Y 35.7031, Z -2.1667, A 0.000, B 0.000, C 0.000 }
gfCNCPoint2[4023] = {X 526.5648, Y 35.7893, Z -2.1667, A 0.000, B 0.000, C 0.000 }
gfCNCPoint2[4024] = {X 525.8868, Y 35.7894, Z -2.1667, A 0.000, B 0.000, C 0.000 }
gfCNCPoint2[4025] = {X 524.9433, Y 35.6831, Z -2.1667, A 0.000, B 0.000, C 0.000 }
gfCNCPoint2[4026] = {X 524.0471, Y 35.3696, Z -2.1667, A 0.000, B 0.000, C 0.000 }
gfCNCPoint2[4027] = {X 523.2432, Y 34.8644, Z -2.1667, A 0.000, B 0.000, C 0.000 }
gfCNCPoint2[4028] = {X 522.5718, Y 34.1930, Z -2.1667, A 0.000, B 0.000, C 0.000 }
gfCNCPoint2[4029] = {X 522.0666, Y 33.3891, Z -2.1667, A 0.000, B 0.000, C 0.000 }
gfCNCPoint2[4030] = {X 521.7531, Y 32.4929, Z -2.1667, A 0.000, B 0.000, C 0.000 }
gfCNCPoint2[4031] = {X 521.6468, Y 31.5495, Z -2.1667, A 0.000, B 0.000, C 0.000 }
gfCNCPoint2[4032] = {X 521.6468, Y 24.5714, Z -2.1667, A 0.000, B 0.000, C 0.000 }
gfCNCPoint2[4033] = {X 521.7519, Y 23.6330, Z -2.1667, A 0.000, B 0.000, C 0.000 }
gfCNCPoint2[4034] = {X 522.0622, Y 22.7411, Z -2.1667, A 0.000, B 0.000, C 0.000 }
gfCNCPoint2[4035] = {X 522.5621, Y 21.9400, Z -2.1667, A 0.000, B 0.000, C 0.000 }
gfCNCPoint2[4036] = {X 523.2270, Y 21.2694, Z -2.1667, A 0.000, B 0.000, C 0.000 }
gfCNCPoint2[4037] = {X 524.0238, Y 20.7626, Z -2.1667, A 0.000, B 0.000, C 0.000 }
gfCNCPoint2[4038] = {X 524.9130, Y 20.4448, Z -2.1667, A 0.000, B 0.000, C 0.000 }
gfCNCPoint2[4039] = {X 525.8505, Y 20.3316, Z -2.1667, A 0.000, B 0.000, C 0.000 }
gfCNCPoint2[4040] = {X 526.5687, Y 20.3316, Z -2.1667, A 0.000, B 0.000, C 0.000 }
gfCNCPoint2[4041] = {X 527.3869, Y 20.4193, Z -2.1667, A 0.000, B 0.000, C 0.000 }
gfCNCPoint2[4042] = {X 528.1728, Y 20.6633, Z -2.1667, A 0.000, B 0.000, C 0.000 }
gfCNCPoint2[4043] = {X 528.8968, Y 21.0545, Z -2.1667, A 0.000, B 0.000, C 0.000 }
gfCNCPoint2[4044] = {X 529.5315, Y 21.5782, Z -2.1667, A 0.000, B 0.000, C 0.000 }
gfCNCPoint2[4045] = {X 530.0531, Y 22.2147, Z -2.1667, A 0.000, B 0.000, C 0.000 }
gfCNCPoint2[4046] = {X 534.7119, Y 22.2151, Z -2.1667, A 0.000, B 0.000, C 0.000 }
gfCNCPoint2[4047] = {X 534.7119, Y 19.6212, Z -2.1667, A 0.000, B 0.000, C 0.000 }
gfCNCPoint2[4048] = {X 524.1495, Y 19.6207, Z -2.1667, A 0.000, B 0.000, C 0.000 }
gfCNCPoint2[4049] = {X 524.1264, Y 19.6560, Z -2.1667, A 0.000, B 0.000, C 0.000 }
gfCNCPoint2[4050] = {X 523.6038, Y 20.2889, Z -2.1667, A 0.000, B 0.000, C 0.000 }
gfCNCPoint2[4051] = {X 522.9691, Y 20.8094, Z -2.1667, A 0.000, B 0.000, C 0.000 }
gfCNCPoint2[4052] = {X 522.2460, Y 21.1977, Z -2.1667, A 0.000, B 0.000, C 0.000 }
gfCNCPoint2[4053] = {X 521.4616, Y 21.4395, Z -2.1667, A 0.000, B 0.000, C 0.000 }
gfCNCPoint2[4054] = {X 520.6453, Y 21.5256, Z -2.1667, A 0.000, B 0.000, C 0.000 }
gfCNCPoint2[4055] = {X 519.9691, Y 21.5257, Z -2.1667, A 0.000, B 0.000, C 0.000 }
gfCNCPoint2[4056] = {X 519.0256, Y 21.4194, Z -2.1667, A 0.000, B 0.000, C 0.000 }
gfCNCPoint2[4057] = {X 518.1294, Y 21.1058, Z -2.1667, A 0.000, B 0.000, C 0.000 }
gfCNCPoint2[4058] = {X 517.3255, Y 20.6007, Z -2.1667, A 0.000, B 0.000, C 0.000 }
gfCNCPoint2[4059] = {X 516.6541, Y 19.9293, Z -2.1667, A 0.000, B 0.000, C 0.000 }
gfCNCPoint2[4060] = {X 516.1490, Y 19.1254, Z -2.1667, A 0.000, B 0.000, C 0.000 }
gfCNCPoint2[4061] = {X 515.8354, Y 18.2292, Z -2.1667, A 0.000, B 0.000, C 0.000 }
gfCNCPoint2[4062] = {X 515.7291, Y 17.2857, Z -2.1667, A 0.000, B 0.000, C 0.000 }
gfCNCPoint2[4063] = {X 515.7291, Y 10.3077, Z -2.1667, A 0.000, B 0.000, C 0.000 }
gfCNCPoint2[4064] = {X 515.8342, Y 9.3696, Z -2.1667, A 0.000, B 0.000, C 0.000 }
gfCNCPoint2[4065] = {X 516.1442, Y 8.4780, Z -2.1667, A 0.000, B 0.000, C 0.000 }
gfCNCPoint2[4066] = {X 516.6438, Y 7.6771, Z -2.1667, A 0.000, B 0.000, C 0.000 }
gfCNCPoint2[4067] = {X 517.3082, Y 7.0066, Z -2.1667, A 0.000, B 0.000, C 0.000 }
gfCNCPoint2[4068] = {X 518.1045, Y 6.4997, Z -2.1667, A 0.000, B 0.000, C 0.000 }
gfCNCPoint2[4069] = {X 518.9932, Y 6.1815, Z -2.1667, A 0.000, B 0.000, C 0.000 }
gfCNCPoint2[4070] = {X 519.9303, Y 6.0679, Z -2.1667, A 0.000, B 0.000, C 0.000 }
gfCNCPoint2[4071] = {X 520.6494, Y 6.0679, Z -2.1667, A 0.000, B 0.000, C 0.000 }
gfCNCPoint2[4072] = {X 521.4680, Y 6.1553, Z -2.1667, A 0.000, B 0.000, C 0.000 }
gfCNCPoint2[4073] = {X 522.2543, Y 6.3992, Z -2.1667, A 0.000, B 0.000, C 0.000 }
gfCNCPoint2[4074] = {X 522.9786, Y 6.7904, Z -2.1667, A 0.000, B 0.000, C 0.000 }
gfCNCPoint2[4075] = {X 523.6136, Y 7.3143, Z -2.1667, A 0.000, B 0.000, C 0.000 }
gfCNCPoint2[4076] = {X 524.1355, Y 7.9510, Z -2.1667, A 0.000, B 0.000, C 0.000 }
gfCNCPoint2[4077] = {X 533.9640, Y 7.9513, Z -2.1667, A 0.000, B 0.000, C 0.000 }
gfCNCPoint2[4078] = {X 533.9641, Y 3.9513, Z -2.1667, A 0.000, B 0.000, C 0.000 }
gfCNCPoint2[4079] = {X 533.9640, Y 8.0313, Z -2.1667, A 0.000, B 0.000, C 0.000 }
gfCNCPoint2[4080] = {X 543.7521, Y 8.0316, Z -2.1667, A 0.000, B 0.000, C 0.000 }
gfCNCPoint2[4081] = {X 544.6963, Y 8.1135, Z -2.1667, A 0.000, B 0.000, C 0.000 }
gfCNCPoint2[4082] = {X 545.5974, Y 8.4068, Z -2.1667, A 0.000, B 0.000, C 0.000 }
gfCNCPoint2[4083] = {X 546.4090, Y 8.8961, Z -2.1667, A 0.000, B 0.000, C 0.000 }
gfCNCPoint2[4084] = {X 547.0889, Y 9.5563, Z -2.1667, A 0.000, B 0.000, C 0.000 }
gfCNCPoint2[4085] = {X 547.6020, Y 10.3531, Z -2.1667, A 0.000, B 0.000, C 0.000 }
gfCNCPoint2[4086] = {X 547.9217, Y 11.2452, Z -2.1667, A 0.000, B 0.000, C 0.000 }
gfCNCPoint2[4087] = {X 548.0314, Y 12.1866, Z -2.1667, A 0.000, B 0.000, C 0.000 }
gfCNCPoint2[4088] = {X 548.0312, Y 13.0208, Z -2.1667, A 0.000, B 0.000, C 0.000 }
gfCNCPoint2[4089] = {X 547.9287, Y 13.8967, Z -2.1667, A 0.000, B 0.000, C 0.000 }
gfCNCPoint2[4090] = {X 547.6439, Y 14.7312, Z -2.1667, A 0.000, B 0.000, C 0.000 }
gfCNCPoint2[4091] = {X 547.1897, Y 15.4870, Z -2.1667, A 0.000, B 0.000, C 0.000 }
gfCNCPoint2[4092] = {X 546.5863, Y 16.1300, Z -2.1667, A 0.000, B 0.000, C 0.000 }
gfCNCPoint2[4093] = {X 546.5029, Y 16.2000, Z -2.1667, A 0.000, B 0.000, C 0.000 }
gfCNCPoint2[4094] = {X 546.5031, Y 40.9896, Z -2.1667, A 0.000, B 0.000, C 0.000 }
gfCNCPoint2[4095] = {X 546.5831, Y 41.0541, Z -2.1667, A 0.000, B 0.000, C 0.000 }
gfCNCPoint2[4096] = {X 547.1891, Y 41.6991, Z -2.1667, A 0.000, B 0.000, C 0.000 }
gfCNCPoint2[4097] = {X 547.6449, Y 42.4576, Z -2.1667, A 0.000, B 0.000, C 0.000 }
gfCNCPoint2[4098] = {X 547.9299, Y 43.2955, Z -2.1667, A 0.000, B 0.000, C 0.000 }
gfCNCPoint2[4099] = {X 548.0313, Y 44.1746, Z -2.1667, A 0.000, B 0.000, C 0.000 }
gfCNCPoint2[4100] = {X 548.0314, Y 45.0003, Z -2.1667, A 0.000, B 0.000, C 0.000 }
gfCNCPoint2[4101] = {X 547.9217, Y 45.9416, Z -2.1667, A 0.000, B 0.000, C 0.000 }
gfCNCPoint2[4102] = {X 547.6020, Y 46.8337, Z -2.1667, A 0.000, B 0.000, C 0.000 }
gfCNCPoint2[4103] = {X 547.0889, Y 47.6304, Z -2.1667, A 0.000, B 0.000, C 0.000 }
gfCNCPoint2[4104] = {X 546.4090, Y 48.2906, Z -2.1667, A 0.000, B 0.000, C 0.000 }
gfCNCPoint2[4105] = {X 545.5974, Y 48.7799, Z -2.1667, A 0.000, B 0.000, C 0.000 }
gfCNCPoint2[4106] = {X 544.6962, Y 49.0731, Z -2.1667, A 0.000, B 0.000, C 0.000 }
gfCNCPoint2[4107] = {X 543.7521, Y 49.1549, Z -2.1667, A 0.000, B 0.000, C 0.000 }
gfCNCPoint2[4108] = {X 523.9612, Y 49.1555, Z -2.1667, A 0.000, B 0.000, C 0.000 }
gfCNCPoint2[4109] = {X 523.4345, Y 49.7881, Z -2.1667, A 0.000, B 0.000, C 0.000 }
gfCNCPoint2[4110] = {X 522.7973, Y 50.3092, Z -2.1667, A 0.000, B 0.000, C 0.000 }
gfCNCPoint2[4111] = {X 522.0729, Y 50.7000, Z -2.1667, A 0.000, B 0.000, C 0.000 }
gfCNCPoint2[4112] = {X 521.2874, Y 50.9463, Z -2.1667, A 0.000, B 0.000, C 0.000 }
gfCNCPoint2[4113] = {X 520.4695, Y 51.0391, Z -2.1667, A 0.000, B 0.000, C 0.000 }
gfCNCPoint2[4114] = {X 519.7998, Y 51.0391, Z -2.1667, A 0.000, B 0.000, C 0.000 }
gfCNCPoint2[4115] = {X 518.8741, Y 50.9348, Z -2.1667, A 0.000, B 0.000, C 0.000 }
gfCNCPoint2[4116] = {X 517.9948, Y 50.6272, Z -2.1667, A 0.000, B 0.000, C 0.000 }
gfCNCPoint2[4117] = {X 517.2061, Y 50.1315, Z -2.1667, A 0.000, B 0.000, C 0.000 }
gfCNCPoint2[4118] = {X 516.5474, Y 49.4728, Z -2.1667, A 0.000, B 0.000, C 0.000 }
gfCNCPoint2[4119] = {X 516.0517, Y 48.6841, Z -2.1667, A 0.000, B 0.000, C 0.000 }
gfCNCPoint2[4120] = {X 515.7441, Y 47.8048, Z -2.1667, A 0.000, B 0.000, C 0.000 }
gfCNCPoint2[4121] = {X 515.6398, Y 46.8791, Z -2.1667, A 0.000, B 0.000, C 0.000 }
gfCNCPoint2[4122] = {X 515.6398, Y 39.9011, Z -2.1667, A 0.000, B 0.000, C 0.000 }
gfCNCPoint2[4123] = {X 515.7429, Y 38.9805, Z -2.1667, A 0.000, B 0.000, C 0.000 }
gfCNCPoint2[4124] = {X 516.0472, Y 38.1056, Z -2.1667, A 0.000, B 0.000, C 0.000 }
gfCNCPoint2[4125] = {X 516.5376, Y 37.3197, Z -2.1667, A 0.000, B 0.000, C 0.000 }
gfCNCPoint2[4126] = {X 517.1897, Y 36.6618, Z -2.1667, A 0.000, B 0.000, C 0.000 }
gfCNCPoint2[4127] = {X 517.9713, Y 36.1645, Z -2.1667, A 0.000, B 0.000, C 0.000 }
gfCNCPoint2[4128] = {X 518.8435, Y 35.8525, Z -2.1667, A 0.000, B 0.000, C 0.000 }
gfCNCPoint2[4129] = {X 519.7631, Y 35.7413, Z -2.1667, A 0.000, B 0.000, C 0.000 }
gfCNCPoint2[4130] = {X 520.5247, Y 35.7415, Z -2.1667, A 0.000, B 0.000, C 0.000 }
gfCNCPoint2[4131] = {X 521.3373, Y 35.8329, Z -2.1667, A 0.000, B 0.000, C 0.000 }
gfCNCPoint2[4132] = {X 522.1163, Y 36.0815, Z -2.1667, A 0.000, B 0.000, C 0.000 }
gfCNCPoint2[4133] = {X 522.8316, Y 36.4777, Z -2.1667, A 0.000, B 0.000, C 0.000 }
gfCNCPoint2[4134] = {X 523.4557, Y 37.0062, Z -2.1667, A 0.000, B 0.000, C 0.000 }
gfCNCPoint2[4135] = {X 523.9642, Y 37.6465, Z -2.1667, A 0.000, B 0.000, C 0.000 }
gfCNCPoint2[4136] = {X 534.7919, Y 37.6471, Z -2.1667, A 0.000, B 0.000, C 0.000 }
gfCNCPoint2[4137] = {X 534.7919, Y 33.8048, Z -2.1667, A 0.000, B 0.000, C 0.000 }
gfCNCPoint2[4138] = {X 530.0216, Y 33.8042, Z -2.1667, A 0.000, B 0.000, C 0.000 }
gfCNCPoint2[4139] = {X 529.9750, Y 33.8790, Z -2.1667, A 0.000, B 0.000, C 0.000 }
gfCNCPoint2[4140] = {X 529.4625, Y 34.4985, Z -2.1667, A 0.000, B 0.000, C 0.000 }
gfCNCPoint2[4141] = {X 528.8404, Y 35.0078, Z -2.1667, A 0.000, B 0.000, C 0.000 }
gfCNCPoint2[4142] = {X 528.1320, Y 35.3880, Z -2.1667, A 0.000, B 0.000, C 0.000 }
gfCNCPoint2[4143] = {X 527.3636, Y 35.6247, Z -2.1667, A 0.000, B 0.000, C 0.000 }
gfCNCPoint2[4144] = {X 526.5641, Y 35.7093, Z -2.1667, A 0.000, B 0.000, C 0.000 }
gfCNCPoint2[4145] = {X 525.8868, Y 35.7095, Z -2.1667, A 0.000, B 0.000, C 0.000 }
gfCNCPoint2[4146] = {X 524.9611, Y 35.6052, Z -2.1667, A 0.000, B 0.000, C 0.000 }
gfCNCPoint2[4147] = {X 524.0818, Y 35.2975, Z -2.1667, A 0.000, B 0.000, C 0.000 }
gfCNCPoint2[4148] = {X 523.2930, Y 34.8019, Z -2.1667, A 0.000, B 0.000, C 0.000 }
gfCNCPoint2[4149] = {X 522.6343, Y 34.1432, Z -2.1667, A 0.000, B 0.000, C 0.000 }
gfCNCPoint2[4150] = {X 522.1387, Y 33.3544, Z -2.1667, A 0.000, B 0.000, C 0.000 }
gfCNCPoint2[4151] = {X 521.8311, Y 32.4751, Z -2.1667, A 0.000, B 0.000, C 0.000 }
gfCNCPoint2[4152] = {X 521.7268, Y 31.5495, Z -2.1667, A 0.000, B 0.000, C 0.000 }
gfCNCPoint2[4153] = {X 521.7268, Y 24.5714, Z -2.1667, A 0.000, B 0.000, C 0.000 }
gfCNCPoint2[4154] = {X 521.8299, Y 23.6507, Z -2.1667, A 0.000, B 0.000, C 0.000 }
gfCNCPoint2[4155] = {X 522.1343, Y 22.7756, Z -2.1667, A 0.000, B 0.000, C 0.000 }
gfCNCPoint2[4156] = {X 522.6248, Y 21.9897, Z -2.1667, A 0.000, B 0.000, C 0.000 }
gfCNCPoint2[4157] = {X 523.2772, Y 21.3317, Z -2.1667, A 0.000, B 0.000, C 0.000 }
gfCNCPoint2[4158] = {X 524.0589, Y 20.8345, Z -2.1667, A 0.000, B 0.000, C 0.000 }
gfCNCPoint2[4159] = {X 524.9313, Y 20.5226, Z -2.1667, A 0.000, B 0.000, C 0.000 }
gfCNCPoint2[4160] = {X 525.8511, Y 20.4116, Z -2.1667, A 0.000, B 0.000, C 0.000 }
gfCNCPoint2[4161] = {X 526.5679, Y 20.4116, Z -2.1667, A 0.000, B 0.000, C 0.000 }
gfCNCPoint2[4162] = {X 527.3791, Y 20.4993, Z -2.1667, A 0.000, B 0.000, C 0.000 }
gfCNCPoint2[4163] = {X 528.1575, Y 20.7437, Z -2.1667, A 0.000, B 0.000, C 0.000 }
gfCNCPoint2[4164] = {X 528.8732, Y 21.1352, Z -2.1667, A 0.000, B 0.000, C 0.000 }
gfCNCPoint2[4165] = {X 529.4988, Y 21.6589, Z -2.1667, A 0.000, B 0.000, C 0.000 }
gfCNCPoint2[4166] = {X 530.0101, Y 22.2947, Z -2.1667, A 0.000, B 0.000, C 0.000 }
gfCNCPoint2[4167] = {X 534.7919, Y 22.2951, Z -2.1667, A 0.000, B 0.000, C 0.000 }
gfCNCPoint2[4168] = {X 534.7919, Y 19.5412, Z -2.1667, A 0.000, B 0.000, C 0.000 }
gfCNCPoint2[4169] = {X 524.1051, Y 19.5407, Z -2.1667, A 0.000, B 0.000, C 0.000 }
gfCNCPoint2[4170] = {X 524.0766, Y 19.5865, Z -2.1667, A 0.000, B 0.000, C 0.000 }
gfCNCPoint2[4171] = {X 523.5642, Y 20.2154, Z -2.1667, A 0.000, B 0.000, C 0.000 }
gfCNCPoint2[4172] = {X 522.9394, Y 20.7329, Z -2.1667, A 0.000, B 0.000, C 0.000 }
gfCNCPoint2[4173] = {X 522.2261, Y 21.1193, Z -2.1667, A 0.000, B 0.000, C 0.000 }
gfCNCPoint2[4174] = {X 521.4514, Y 21.3599, Z -2.1667, A 0.000, B 0.000, C 0.000 }
gfCNCPoint2[4175] = {X 520.6447, Y 21.4456, Z -2.1667, A 0.000, B 0.000, C 0.000 }
gfCNCPoint2[4176] = {X 519.9691, Y 21.4457, Z -2.1667, A 0.000, B 0.000, C 0.000 }
gfCNCPoint2[4177] = {X 519.0434, Y 21.3414, Z -2.1667, A 0.000, B 0.000, C 0.000 }
gfCNCPoint2[4178] = {X 518.1641, Y 21.0337, Z -2.1667, A 0.000, B 0.000, C 0.000 }
gfCNCPoint2[4179] = {X 517.3754, Y 20.5381, Z -2.1667, A 0.000, B 0.000, C 0.000 }
gfCNCPoint2[4180] = {X 516.7167, Y 19.8794, Z -2.1667, A 0.000, B 0.000, C 0.000 }
gfCNCPoint2[4181] = {X 516.2211, Y 19.0907, Z -2.1667, A 0.000, B 0.000, C 0.000 }
gfCNCPoint2[4182] = {X 515.9134, Y 18.2114, Z -2.1667, A 0.000, B 0.000, C 0.000 }
gfCNCPoint2[4183] = {X 515.8091, Y 17.2857, Z -2.1667, A 0.000, B 0.000, C 0.000 }
gfCNCPoint2[4184] = {X 515.8091, Y 10.3077, Z -2.1667, A 0.000, B 0.000, C 0.000 }
gfCNCPoint2[4185] = {X 515.9122, Y 9.3873, Z -2.1667, A 0.000, B 0.000, C 0.000 }
gfCNCPoint2[4186] = {X 516.2164, Y 8.5125, Z -2.1667, A 0.000, B 0.000, C 0.000 }
gfCNCPoint2[4187] = {X 516.7065, Y 7.7267, Z -2.1667, A 0.000, B 0.000, C 0.000 }
gfCNCPoint2[4188] = {X 517.3584, Y 7.0689, Z -2.1667, A 0.000, B 0.000, C 0.000 }
gfCNCPoint2[4189] = {X 518.1397, Y 6.5715, Z -2.1667, A 0.000, B 0.000, C 0.000 }
gfCNCPoint2[4190] = {X 519.0117, Y 6.2594, Z -2.1667, A 0.000, B 0.000, C 0.000 }
gfCNCPoint2[4191] = {X 519.9311, Y 6.1479, Z -2.1667, A 0.000, B 0.000, C 0.000 }
gfCNCPoint2[4192] = {X 520.6487, Y 6.1479, Z -2.1667, A 0.000, B 0.000, C 0.000 }
gfCNCPoint2[4193] = {X 521.4602, Y 6.2353, Z -2.1667, A 0.000, B 0.000, C 0.000 }
gfCNCPoint2[4194] = {X 522.2390, Y 6.4796, Z -2.1667, A 0.000, B 0.000, C 0.000 }
gfCNCPoint2[4195] = {X 522.9551, Y 6.8711, Z -2.1667, A 0.000, B 0.000, C 0.000 }
gfCNCPoint2[4196] = {X 523.5809, Y 7.3950, Z -2.1667, A 0.000, B 0.000, C 0.000 }
gfCNCPoint2[4197] = {X 524.0925, Y 8.0310, Z -2.1667, A 0.000, B 0.000, C 0.000 }
gfCNCPoint2[4198] = {X 533.9640, Y 8.0313, Z -2.1667, A 0.000, B 0.000, C 0.000 }
gfCNCPoint2[4199] = {X 533.9641, Y 4.0313, Z -2.1667, A 0.000, B 0.000, C 0.000 }
gfCNCPoint2[4200] = {X 533.9640, Y 8.1113, Z -2.1667, A 0.000, B 0.000, C 0.000 }
gfCNCPoint2[4201] = {X 543.7532, Y 8.1116, Z -2.1667, A 0.000, B 0.000, C 0.000 }
gfCNCPoint2[4202] = {X 544.6794, Y 8.1917, Z -2.1667, A 0.000, B 0.000, C 0.000 }
gfCNCPoint2[4203] = {X 545.5635, Y 8.4792, Z -2.1667, A 0.000, B 0.000, C 0.000 }
gfCNCPoint2[4204] = {X 546.3597, Y 8.9591, Z -2.1667, A 0.000, B 0.000, C 0.000 }
gfCNCPoint2[4205] = {X 547.0267, Y 9.6066, Z -2.1667, A 0.000, B 0.000, C 0.000 }
gfCNCPoint2[4206] = {X 547.5301, Y 10.3882, Z -2.1667, A 0.000, B 0.000, C 0.000 }
gfCNCPoint2[4207] = {X 547.8438, Y 11.2633, Z -2.1667, A 0.000, B 0.000, C 0.000 }
gfCNCPoint2[4208] = {X 547.9514, Y 12.1867, Z -2.1667, A 0.000, B 0.000, C 0.000 }
gfCNCPoint2[4209] = {X 547.9512, Y 13.0200, Z -2.1667, A 0.000, B 0.000, C 0.000 }
gfCNCPoint2[4210] = {X 547.8507, Y 13.8790, Z -2.1667, A 0.000, B 0.000, C 0.000 }
gfCNCPoint2[4211] = {X 547.5714, Y 14.6975, Z -2.1667, A 0.000, B 0.000, C 0.000 }
gfCNCPoint2[4212] = {X 547.1258, Y 15.4387, Z -2.1667, A 0.000, B 0.000, C 0.000 }
gfCNCPoint2[4213] = {X 546.5341, Y 16.0694, Z -2.1667, A 0.000, B 0.000, C 0.000 }
gfCNCPoint2[4214] = {X 546.4795, Y 16.1156, Z -2.1667, A 0.000, B 0.000, C 0.000 }
gfCNCPoint2[4215] = {X 546.4242, Y 16.1607, Z -2.1667, A 0.000, B 0.000, C 0.000 }
gfCNCPoint2[4216] = {X 546.4231, Y 41.0279, Z -2.1667, A 0.000, B 0.000, C 0.000 }
gfCNCPoint2[4217] = {X 546.5319, Y 41.1156, Z -2.1667, A 0.000, B 0.000, C 0.000 }
gfCNCPoint2[4218] = {X 547.1259, Y 41.7481, Z -2.1667, A 0.000, B 0.000, C 0.000 }
gfCNCPoint2[4219] = {X 547.5726, Y 42.4919, Z -2.1667, A 0.000, B 0.000, C 0.000 }
gfCNCPoint2[4220] = {X 547.8519, Y 43.3133, Z -2.1667, A 0.000, B 0.000, C 0.000 }
gfCNCPoint2[4221] = {X 547.9513, Y 44.1753, Z -2.1667, A 0.000, B 0.000, C 0.000 }
gfCNCPoint2[4222] = {X 547.9514, Y 45.0001, Z -2.1667, A 0.000, B 0.000, C 0.000 }
gfCNCPoint2[4223] = {X 547.8438, Y 45.9235, Z -2.1667, A 0.000, B 0.000, C 0.000 }
gfCNCPoint2[4224] = {X 547.5301, Y 46.7986, Z -2.1667, A 0.000, B 0.000, C 0.000 }
gfCNCPoint2[4225] = {X 547.0267, Y 47.5801, Z -2.1667, A 0.000, B 0.000, C 0.000 }
gfCNCPoint2[4226] = {X 546.3597, Y 48.2276, Z -2.1667, A 0.000, B 0.000, C 0.000 }
gfCNCPoint2[4227] = {X 545.5635, Y 48.7074, Z -2.1667, A 0.000, B 0.000, C 0.000 }
gfCNCPoint2[4228] = {X 544.6794, Y 48.9949, Z -2.1667, A 0.000, B 0.000, C 0.000 }
gfCNCPoint2[4229] = {X 543.7532, Y 49.0749, Z -2.1667, A 0.000, B 0.000, C 0.000 }
gfCNCPoint2[4230] = {X 523.9187, Y 49.0755, Z -2.1667, A 0.000, B 0.000, C 0.000 }
gfCNCPoint2[4231] = {X 523.4021, Y 49.7073, Z -2.1667, A 0.000, B 0.000, C 0.000 }
gfCNCPoint2[4232] = {X 522.7740, Y 50.2285, Z -2.1667, A 0.000, B 0.000, C 0.000 }
gfCNCPoint2[4233] = {X 522.0576, Y 50.6196, Z -2.1667, A 0.000, B 0.000, C 0.000 }
gfCNCPoint2[4234] = {X 521.2796, Y 50.8662, Z -2.1667, A 0.000, B 0.000, C 0.000 }
gfCNCPoint2[4235] = {X 520.4688, Y 50.9591, Z -2.1667, A 0.000, B 0.000, C 0.000 }
gfCNCPoint2[4236] = {X 519.7998, Y 50.9591, Z -2.1667, A 0.000, B 0.000, C 0.000 }
gfCNCPoint2[4237] = {X 518.8919, Y 50.8568, Z -2.1667, A 0.000, B 0.000, C 0.000 }
gfCNCPoint2[4238] = {X 518.0295, Y 50.5551, Z -2.1667, A 0.000, B 0.000, C 0.000 }
gfCNCPoint2[4239] = {X 517.2559, Y 50.0690, Z -2.1667, A 0.000, B 0.000, C 0.000 }
gfCNCPoint2[4240] = {X 516.6099, Y 49.4230, Z -2.1667, A 0.000, B 0.000, C 0.000 }
gfCNCPoint2[4241] = {X 516.1238, Y 48.6494, Z -2.1667, A 0.000, B 0.000, C 0.000 }
gfCNCPoint2[4242] = {X 515.8221, Y 47.7870, Z -2.1667, A 0.000, B 0.000, C 0.000 }
gfCNCPoint2[4243] = {X 515.7198, Y 46.8791, Z -2.1667, A 0.000, B 0.000, C 0.000 }
gfCNCPoint2[4244] = {X 515.7198, Y 39.9011, Z -2.1667, A 0.000, B 0.000, C 0.000 }
gfCNCPoint2[4245] = {X 515.8209, Y 38.9982, Z -2.1667, A 0.000, B 0.000, C 0.000 }
gfCNCPoint2[4246] = {X 516.1194, Y 38.1401, Z -2.1667, A 0.000, B 0.000, C 0.000 }
gfCNCPoint2[4247] = {X 516.6003, Y 37.3693, Z -2.1667, A 0.000, B 0.000, C 0.000 }
gfCNCPoint2[4248] = {X 517.2399, Y 36.7241, Z -2.1667, A 0.000, B 0.000, C 0.000 }
gfCNCPoint2[4249] = {X 518.0064, Y 36.2364, Z -2.1667, A 0.000, B 0.000, C 0.000 }
gfCNCPoint2[4250] = {X 518.8619, Y 35.9304, Z -2.1667, A 0.000, B 0.000, C 0.000 }
gfCNCPoint2[4251] = {X 519.7638, Y 35.8213, Z -2.1667, A 0.000, B 0.000, C 0.000 }
gfCNCPoint2[4252] = {X 520.5236, Y 35.8215, Z -2.1667, A 0.000, B 0.000, C 0.000 }
gfCNCPoint2[4253] = {X 521.3291, Y 35.9130, Z -2.1667, A 0.000, B 0.000, C 0.000 }
gfCNCPoint2[4254] = {X 522.1006, Y 36.1619, Z -2.1667, A 0.000, B 0.000, C 0.000 }
gfCNCPoint2[4255] = {X 522.8076, Y 36.5584, Z -2.1667, A 0.000, B 0.000, C 0.000 }
gfCNCPoint2[4256] = {X 523.4223, Y 37.0869, Z -2.1667, A 0.000, B 0.000, C 0.000 }
gfCNCPoint2[4257] = {X 523.9204, Y 37.7265, Z -2.1667, A 0.000, B 0.000, C 0.000 }
gfCNCPoint2[4258] = {X 534.8719, Y 37.7271, Z -2.1667, A 0.000, B 0.000, C 0.000 }
gfCNCPoint2[4259] = {X 534.8719, Y 33.7248, Z -2.1667, A 0.000, B 0.000, C 0.000 }
gfCNCPoint2[4260] = {X 529.9773, Y 33.7242, Z -2.1667, A 0.000, B 0.000, C 0.000 }
gfCNCPoint2[4261] = {X 529.9071, Y 33.8366, Z -2.1667, A 0.000, B 0.000, C 0.000 }
gfCNCPoint2[4262] = {X 529.2612, Y 34.5790, Z -2.1667, A 0.000, B 0.000, C 0.000 }
gfCNCPoint2[4263] = {X 528.4563, Y 35.1452, Z -2.1667, A 0.000, B 0.000, C 0.000 }
gfCNCPoint2[4264] = {X 527.5392, Y 35.5023, Z -2.1667, A 0.000, B 0.000, C 0.000 }
gfCNCPoint2[4265] = {X 526.5634, Y 35.6293, Z -2.1667, A 0.000, B 0.000, C 0.000 }
gfCNCPoint2[4266] = {X 525.8868, Y 35.6295, Z -2.1667, A 0.000, B 0.000, C 0.000 }
gfCNCPoint2[4267] = {X 524.9789, Y 35.5272, Z -2.1667, A 0.000, B 0.000, C 0.000 }
gfCNCPoint2[4268] = {X 524.1165, Y 35.2254, Z -2.1667, A 0.000, B 0.000, C 0.000 }
gfCNCPoint2[4269] = {X 523.3429, Y 34.7393, Z -2.1667, A 0.000, B 0.000, C 0.000 }
gfCNCPoint2[4270] = {X 522.6969, Y 34.0933, Z -2.1667, A 0.000, B 0.000, C 0.000 }
gfCNCPoint2[4271] = {X 522.2108, Y 33.3197, Z -2.1667, A 0.000, B 0.000, C 0.000 }
gfCNCPoint2[4272] = {X 521.9091, Y 32.4573, Z -2.1667, A 0.000, B 0.000, C 0.000 }
gfCNCPoint2[4273] = {X 521.8068, Y 31.5495, Z -2.1667, A 0.000, B 0.000, C 0.000 }
gfCNCPoint2[4274] = {X 521.8068, Y 24.5714, Z -2.1667, A 0.000, B 0.000, C 0.000 }
gfCNCPoint2[4275] = {X 521.9079, Y 23.6684, Z -2.1667, A 0.000, B 0.000, C 0.000 }
gfCNCPoint2[4276] = {X 522.2065, Y 22.8102, Z -2.1667, A 0.000, B 0.000, C 0.000 }
gfCNCPoint2[4277] = {X 522.6876, Y 22.0393, Z -2.1667, A 0.000, B 0.000, C 0.000 }
gfCNCPoint2[4278] = {X 523.3273, Y 21.3940, Z -2.1667, A 0.000, B 0.000, C 0.000 }
gfCNCPoint2[4279] = {X 524.0941, Y 20.9064, Z -2.1667, A 0.000, B 0.000, C 0.000 }
gfCNCPoint2[4280] = {X 524.9497, Y 20.6005, Z -2.1667, A 0.000, B 0.000, C 0.000 }
gfCNCPoint2[4281] = {X 525.8518, Y 20.4916, Z -2.1667, A 0.000, B 0.000, C 0.000 }
gfCNCPoint2[4282] = {X 526.5672, Y 20.4916, Z -2.1667, A 0.000, B 0.000, C 0.000 }
gfCNCPoint2[4283] = {X 527.3712, Y 20.5794, Z -2.1667, A 0.000, B 0.000, C 0.000 }
gfCNCPoint2[4284] = {X 528.1420, Y 20.8241, Z -2.1667, A 0.000, B 0.000, C 0.000 }
gfCNCPoint2[4285] = {X 528.8495, Y 21.2159, Z -2.1667, A 0.000, B 0.000, C 0.000 }
gfCNCPoint2[4286] = {X 529.4657, Y 21.7397, Z -2.1667, A 0.000, B 0.000, C 0.000 }
gfCNCPoint2[4287] = {X 529.9666, Y 22.3747, Z -2.1667, A 0.000, B 0.000, C 0.000 }
gfCNCPoint2[4288] = {X 534.8719, Y 22.3751, Z -2.1667, A 0.000, B 0.000, C 0.000 }
gfCNCPoint2[4289] = {X 534.8719, Y 19.4612, Z -2.1667, A 0.000, B 0.000, C 0.000 }
gfCNCPoint2[4290] = {X 524.0607, Y 19.4607, Z -2.1667, A 0.000, B 0.000, C 0.000 }
gfCNCPoint2[4291] = {X 524.0087, Y 19.5442, Z -2.1667, A 0.000, B 0.000, C 0.000 }
gfCNCPoint2[4292] = {X 523.5061, Y 20.1604, Z -2.1667, A 0.000, B 0.000, C 0.000 }
gfCNCPoint2[4293] = {X 522.8935, Y 20.6674, Z -2.1667, A 0.000, B 0.000, C 0.000 }
gfCNCPoint2[4294] = {X 522.1942, Y 21.0459, Z -2.1667, A 0.000, B 0.000, C 0.000 }
gfCNCPoint2[4295] = {X 521.4348, Y 21.2816, Z -2.1667, A 0.000, B 0.000, C 0.000 }
gfCNCPoint2[4296] = {X 520.6440, Y 21.3656, Z -2.1667, A 0.000, B 0.000, C 0.000 }
gfCNCPoint2[4297] = {X 519.9691, Y 21.3657, Z -2.1667, A 0.000, B 0.000, C 0.000 }
gfCNCPoint2[4298] = {X 519.0612, Y 21.2634, Z -2.1667, A 0.000, B 0.000, C 0.000 }
gfCNCPoint2[4299] = {X 518.1989, Y 20.9617, Z -2.1667, A 0.000, B 0.000, C 0.000 }
gfCNCPoint2[4300] = {X 517.4253, Y 20.4756, Z -2.1667, A 0.000, B 0.000, C 0.000 }
gfCNCPoint2[4301] = {X 516.7792, Y 19.8296, Z -2.1667, A 0.000, B 0.000, C 0.000 }
gfCNCPoint2[4302] = {X 516.2932, Y 19.0560, Z -2.1667, A 0.000, B 0.000, C 0.000 }
gfCNCPoint2[4303] = {X 515.9914, Y 18.1936, Z -2.1667, A 0.000, B 0.000, C 0.000 }
gfCNCPoint2[4304] = {X 515.8891, Y 17.2857, Z -2.1667, A 0.000, B 0.000, C 0.000 }
gfCNCPoint2[4305] = {X 515.8891, Y 10.3077, Z -2.1667, A 0.000, B 0.000, C 0.000 }
gfCNCPoint2[4306] = {X 515.9902, Y 9.4050, Z -2.1667, A 0.000, B 0.000, C 0.000 }
gfCNCPoint2[4307] = {X 516.2885, Y 8.5471, Z -2.1667, A 0.000, B 0.000, C 0.000 }
gfCNCPoint2[4308] = {X 516.7693, Y 7.7764, Z -2.1667, A 0.000, B 0.000, C 0.000 }
gfCNCPoint2[4309] = {X 517.4086, Y 7.1312, Z -2.1667, A 0.000, B 0.000, C 0.000 }
gfCNCPoint2[4310] = {X 518.1749, Y 6.6434, Z -2.1667, A 0.000, B 0.000, C 0.000 }
gfCNCPoint2[4311] = {X 519.0301, Y 6.3372, Z -2.1667, A 0.000, B 0.000, C 0.000 }
gfCNCPoint2[4312] = {X 519.9318, Y 6.2279, Z -2.1667, A 0.000, B 0.000, C 0.000 }
gfCNCPoint2[4313] = {X 520.6480, Y 6.2279, Z -2.1667, A 0.000, B 0.000, C 0.000 }
gfCNCPoint2[4314] = {X 521.4523, Y 6.3154, Z -2.1667, A 0.000, B 0.000, C 0.000 }
gfCNCPoint2[4315] = {X 522.2235, Y 6.5600, Z -2.1667, A 0.000, B 0.000, C 0.000 }
gfCNCPoint2[4316] = {X 522.9313, Y 6.9519, Z -2.1667, A 0.000, B 0.000, C 0.000 }
gfCNCPoint2[4317] = {X 523.5479, Y 7.4758, Z -2.1667, A 0.000, B 0.000, C 0.000 }
gfCNCPoint2[4318] = {X 524.0489, Y 8.1110, Z -2.1667, A 0.000, B 0.000, C 0.000 }
gfCNCPoint2[4319] = {X 533.9640, Y 8.1113, Z -2.1667, A 0.000, B 0.000, C 0.000 }
gfCNCPoint2[4320] = {X 533.9641, Y 4.1113, Z -2.1667, A 0.000, B 0.000, C 0.000 }
gfCNCPoint2[4321] = {X 533.9639, Y 8.1913, Z -2.1667, A 0.000, B 0.000, C 0.000 }
gfCNCPoint2[4322] = {X 543.7544, Y 8.1916, Z -2.1667, A 0.000, B 0.000, C 0.000 }
gfCNCPoint2[4323] = {X 544.6626, Y 8.2699, Z -2.1667, A 0.000, B 0.000, C 0.000 }
gfCNCPoint2[4324] = {X 545.5295, Y 8.5516, Z -2.1667, A 0.000, B 0.000, C 0.000 }
gfCNCPoint2[4325] = {X 546.3104, Y 9.0221, Z -2.1667, A 0.000, B 0.000, C 0.000 }
gfCNCPoint2[4326] = {X 546.9646, Y 9.6570, Z -2.1667, A 0.000, B 0.000, C 0.000 }
gfCNCPoint2[4327] = {X 547.4582, Y 10.4233, Z -2.1667, A 0.000, B 0.000, C 0.000 }
gfCNCPoint2[4328] = {X 547.7658, Y 11.2814, Z -2.1667, A 0.000, B 0.000, C 0.000 }
gfCNCPoint2[4329] = {X 547.8714, Y 12.1869, Z -2.1667, A 0.000, B 0.000, C 0.000 }
gfCNCPoint2[4330] = {X 547.8712, Y 13.0192, Z -2.1667, A 0.000, B 0.000, C 0.000 }
gfCNCPoint2[4331] = {X 547.7727, Y 13.8613, Z -2.1667, A 0.000, B 0.000, C 0.000 }
gfCNCPoint2[4332] = {X 547.4989, Y 14.6638, Z -2.1667, A 0.000, B 0.000, C 0.000 }
gfCNCPoint2[4333] = {X 547.0620, Y 15.3905, Z -2.1667, A 0.000, B 0.000, C 0.000 }
gfCNCPoint2[4334] = {X 546.4819, Y 16.0088, Z -2.1667, A 0.000, B 0.000, C 0.000 }
gfCNCPoint2[4335] = {X 546.4144, Y 16.0656, Z -2.1667, A 0.000, B 0.000, C 0.000 }
gfCNCPoint2[4336] = {X 546.3458, Y 16.1209, Z -2.1667, A 0.000, B 0.000, C 0.000 }
gfCNCPoint2[4337] = {X 546.3429, Y 16.3119, Z -2.1667, A 0.000, B 0.000, C 0.000 }
gfCNCPoint2[4338] = {X 546.3431, Y 41.0662, Z -2.1667, A 0.000, B 0.000, C 0.000 }
gfCNCPoint2[4339] = {X 546.4821, Y 41.1782, Z -2.1667, A 0.000, B 0.000, C 0.000 }
gfCNCPoint2[4340] = {X 547.0684, Y 41.8047, Z -2.1667, A 0.000, B 0.000, C 0.000 }
gfCNCPoint2[4341] = {X 547.5076, Y 42.5419, Z -2.1667, A 0.000, B 0.000, C 0.000 }
gfCNCPoint2[4342] = {X 547.7794, Y 43.3558, Z -2.1667, A 0.000, B 0.000, C 0.000 }
gfCNCPoint2[4343] = {X 547.8714, Y 44.2089, Z -2.1667, A 0.000, B 0.000, C 0.000 }
gfCNCPoint2[4344] = {X 547.8714, Y 44.9999, Z -2.1667, A 0.000, B 0.000, C 0.000 }
gfCNCPoint2[4345] = {X 547.7658, Y 45.9054, Z -2.1667, A 0.000, B 0.000, C 0.000 }
gfCNCPoint2[4346] = {X 547.4582, Y 46.7635, Z -2.1667, A 0.000, B 0.000, C 0.000 }
gfCNCPoint2[4347] = {X 546.9645, Y 47.5298, Z -2.1667, A 0.000, B 0.000, C 0.000 }
gfCNCPoint2[4348] = {X 546.3103, Y 48.1646, Z -2.1667, A 0.000, B 0.000, C 0.000 }
gfCNCPoint2[4349] = {X 545.5295, Y 48.6350, Z -2.1667, A 0.000, B 0.000, C 0.000 }
gfCNCPoint2[4350] = {X 544.6626, Y 48.9166, Z -2.1667, A 0.000, B 0.000, C 0.000 }
gfCNCPoint2[4351] = {X 543.7544, Y 48.9949, Z -2.1667, A 0.000, B 0.000, C 0.000 }
gfCNCPoint2[4352] = {X 523.8756, Y 48.9955, Z -2.1667, A 0.000, B 0.000, C 0.000 }
gfCNCPoint2[4353] = {X 523.3693, Y 49.6266, Z -2.1667, A 0.000, B 0.000, C 0.000 }
gfCNCPoint2[4354] = {X 522.7504, Y 50.1477, Z -2.1667, A 0.000, B 0.000, C 0.000 }
gfCNCPoint2[4355] = {X 522.0423, Y 50.5391, Z -2.1667, A 0.000, B 0.000, C 0.000 }
gfCNCPoint2[4356] = {X 521.2718, Y 50.7861, Z -2.1667, A 0.000, B 0.000, C 0.000 }
gfCNCPoint2[4357] = {X 520.4681, Y 50.8791, Z -2.1667, A 0.000, B 0.000, C 0.000 }
gfCNCPoint2[4358] = {X 519.7998, Y 50.8791, Z -2.1667, A 0.000, B 0.000, C 0.000 }
gfCNCPoint2[4359] = {X 518.9097, Y 50.7788, Z -2.1667, A 0.000, B 0.000, C 0.000 }
gfCNCPoint2[4360] = {X 518.0642, Y 50.4830, Z -2.1667, A 0.000, B 0.000, C 0.000 }
gfCNCPoint2[4361] = {X 517.3058, Y 50.0064, Z -2.1667, A 0.000, B 0.000, C 0.000 }
gfCNCPoint2[4362] = {X 516.6724, Y 49.3731, Z -2.1667, A 0.000, B 0.000, C 0.000 }
gfCNCPoint2[4363] = {X 516.1959, Y 48.6147, Z -2.1667, A 0.000, B 0.000, C 0.000 }
gfCNCPoint2[4364] = {X 515.9001, Y 47.7692, Z -2.1667, A 0.000, B 0.000, C 0.000 }
gfCNCPoint2[4365] = {X 515.7998, Y 46.8791, Z -2.1667, A 0.000, B 0.000, C 0.000 }
gfCNCPoint2[4366] = {X 515.7998, Y 39.9011, Z -2.1667, A 0.000, B 0.000, C 0.000 }
gfCNCPoint2[4367] = {X 515.9001, Y 39.0110, Z -2.1667, A 0.000, B 0.000, C 0.000 }
gfCNCPoint2[4368] = {X 516.1959, Y 38.1655, Z -2.1667, A 0.000, B 0.000, C 0.000 }
gfCNCPoint2[4369] = {X 516.6725, Y 37.4071, Z -2.1667, A 0.000, B 0.000, C 0.000 }
gfCNCPoint2[4370] = {X 517.3059, Y 36.7737, Z -2.1667, A 0.000, B 0.000, C 0.000 }
gfCNCPoint2[4371] = {X 518.0643, Y 36.2972, Z -2.1667, A 0.000, B 0.000, C 0.000 }
gfCNCPoint2[4372] = {X 518.9098, Y 36.0014, Z -2.1667, A 0.000, B 0.000, C 0.000 }
gfCNCPoint2[4373] = {X 519.7999, Y 35.9011, Z -2.1667, A 0.000, B 0.000, C 0.000 }
gfCNCPoint2[4374] = {X 520.5225, Y 35.9015, Z -2.1667, A 0.000, B 0.000, C 0.000 }
gfCNCPoint2[4375] = {X 521.3208, Y 35.9930, Z -2.1667, A 0.000, B 0.000, C 0.000 }
gfCNCPoint2[4376] = {X 522.0847, Y 36.2423, Z -2.1667, A 0.000, B 0.000, C 0.000 }
gfCNCPoint2[4377] = {X 522.7833, Y 36.6392, Z -2.1667, A 0.000, B 0.000, C 0.000 }
gfCNCPoint2[4378] = {X 523.3885, Y 37.1677, Z -2.1667, A 0.000, B 0.000, C 0.000 }
gfCNCPoint2[4379] = {X 523.8759, Y 37.8065, Z -2.1667, A 0.000, B 0.000, C 0.000 }
gfCNCPoint2[4380] = {X 534.9519, Y 37.8071, Z -2.1667, A 0.000, B 0.000, C 0.000 }
gfCNCPoint2[4381] = {X 534.9519, Y 34.0447, Z -2.1667, A 0.000, B 0.000, C 0.000 }
gfCNCPoint2[4382] = {X 534.9531, Y 33.6448, Z -2.1667, A 0.000, B 0.000, C 0.000 }
gfCNCPoint2[4383] = {X 529.9329, Y 33.6442, Z -2.1667, A 0.000, B 0.000, C 0.000 }
gfCNCPoint2[4384] = {X 529.8233, Y 33.8174, Z -2.1667, A 0.000, B 0.000, C 0.000 }
gfCNCPoint2[4385] = {X 529.1838, Y 34.5409, Z -2.1667, A 0.000, B 0.000, C 0.000 }
gfCNCPoint2[4386] = {X 528.3895, Y 35.0901, Z -2.1667, A 0.000, B 0.000, C 0.000 }
gfCNCPoint2[4387] = {X 527.4868, Y 35.4329, Z -2.1667, A 0.000, B 0.000, C 0.000 }
gfCNCPoint2[4388] = {X 526.5283, Y 35.5495, Z -2.1667, A 0.000, B 0.000, C 0.000 }
gfCNCPoint2[4389] = {X 525.8868, Y 35.5495, Z -2.1667, A 0.000, B 0.000, C 0.000 }
gfCNCPoint2[4390] = {X 524.9967, Y 35.4492, Z -2.1667, A 0.000, B 0.000, C 0.000 }
gfCNCPoint2[4391] = {X 524.1512, Y 35.1533, Z -2.1667, A 0.000, B 0.000, C 0.000 }
gfCNCPoint2[4392] = {X 523.3928, Y 34.6768, Z -2.1667, A 0.000, B 0.000, C 0.000 }
gfCNCPoint2[4393] = {X 522.7594, Y 34.0434, Z -2.1667, A 0.000, B 0.000, C 0.000 }
gfCNCPoint2[4394] = {X 522.2829, Y 33.2850, Z -2.1667, A 0.000, B 0.000, C 0.000 }
gfCNCPoint2[4395] = {X 521.9870, Y 32.4395, Z -2.1667, A 0.000, B 0.000, C 0.000 }
gfCNCPoint2[4396] = {X 521.8868, Y 31.5495, Z -2.1667, A 0.000, B 0.000, C 0.000 }
gfCNCPoint2[4397] = {X 521.8868, Y 24.5714, Z -2.1667, A 0.000, B 0.000, C 0.000 }
gfCNCPoint2[4398] = {X 521.9870, Y 23.6813, Z -2.1667, A 0.000, B 0.000, C 0.000 }
gfCNCPoint2[4399] = {X 522.2829, Y 22.8359, Z -2.1667, A 0.000, B 0.000, C 0.000 }
gfCNCPoint2[4400] = {X 522.7594, Y 22.0775, Z -2.1667, A 0.000, B 0.000, C 0.000 }
gfCNCPoint2[4401] = {X 523.3928, Y 21.4441, Z -2.1667, A 0.000, B 0.000, C 0.000 }
gfCNCPoint2[4402] = {X 524.1512, Y 20.9675, Z -2.1667, A 0.000, B 0.000, C 0.000 }
gfCNCPoint2[4403] = {X 524.9967, Y 20.6717, Z -2.1667, A 0.000, B 0.000, C 0.000 }
gfCNCPoint2[4404] = {X 525.8868, Y 20.5714, Z -2.1667, A 0.000, B 0.000, C 0.000 }
gfCNCPoint2[4405] = {X 526.5664, Y 20.5716, Z -2.1667, A 0.000, B 0.000, C 0.000 }
gfCNCPoint2[4406] = {X 527.3632, Y 20.6595, Z -2.1667, A 0.000, B 0.000, C 0.000 }
gfCNCPoint2[4407] = {X 528.1264, Y 20.9045, Z -2.1667, A 0.000, B 0.000, C 0.000 }
gfCNCPoint2[4408] = {X 528.8254, Y 21.2967, Z -2.1667, A 0.000, B 0.000, C 0.000 }
gfCNCPoint2[4409] = {X 529.4322, Y 21.8205, Z -2.1667, A 0.000, B 0.000, C 0.000 }
gfCNCPoint2[4410] = {X 529.9224, Y 22.4547, Z -2.1667, A 0.000, B 0.000, C 0.000 }
gfCNCPoint2[4411] = {X 534.9519, Y 22.4551, Z -2.1667, A 0.000, B 0.000, C 0.000 }
gfCNCPoint2[4412] = {X 534.9519, Y 19.7812, Z -2.1667, A 0.000, B 0.000, C 0.000 }
gfCNCPoint2[4413] = {X 534.9532, Y 19.3812, Z -2.1667, A 0.000, B 0.000, C 0.000 }
gfCNCPoint2[4414] = {X 524.0163, Y 19.3807, Z -2.1667, A 0.000, B 0.000, C 0.000 }
gfCNCPoint2[4415] = {X 523.9055, Y 19.5539, Z -2.1667, A 0.000, B 0.000, C 0.000 }
gfCNCPoint2[4416] = {X 523.2660, Y 20.2773, Z -2.1667, A 0.000, B 0.000, C 0.000 }
gfCNCPoint2[4417] = {X 522.4718, Y 20.8264, Z -2.1667, A 0.000, B 0.000, C 0.000 }
gfCNCPoint2[4418] = {X 521.5692, Y 21.1692, Z -2.1667, A 0.000, B 0.000, C 0.000 }
gfCNCPoint2[4419] = {X 520.6107, Y 21.2857, Z -2.1667, A 0.000, B 0.000, C 0.000 }
gfCNCPoint2[4420] = {X 519.9691, Y 21.2857, Z -2.1667, A 0.000, B 0.000, C 0.000 }
gfCNCPoint2[4421] = {X 519.0790, Y 21.1854, Z -2.1667, A 0.000, B 0.000, C 0.000 }
gfCNCPoint2[4422] = {X 518.2336, Y 20.8896, Z -2.1667, A 0.000, B 0.000, C 0.000 }
gfCNCPoint2[4423] = {X 517.4751, Y 20.4130, Z -2.1667, A 0.000, B 0.000, C 0.000 }
gfCNCPoint2[4424] = {X 516.8418, Y 19.7797, Z -2.1667, A 0.000, B 0.000, C 0.000 }
gfCNCPoint2[4425] = {X 516.3652, Y 19.0212, Z -2.1667, A 0.000, B 0.000, C 0.000 }
gfCNCPoint2[4426] = {X 516.0694, Y 18.1758, Z -2.1667, A 0.000, B 0.000, C 0.000 }
gfCNCPoint2[4427] = {X 515.9691, Y 17.2857, Z -2.1667, A 0.000, B 0.000, C 0.000 }
gfCNCPoint2[4428] = {X 515.9691, Y 10.3077, Z -2.1667, A 0.000, B 0.000, C 0.000 }
gfCNCPoint2[4429] = {X 516.0694, Y 9.4176, Z -2.1667, A 0.000, B 0.000, C 0.000 }
gfCNCPoint2[4430] = {X 516.3652, Y 8.5721, Z -2.1667, A 0.000, B 0.000, C 0.000 }
gfCNCPoint2[4431] = {X 516.8418, Y 7.8137, Z -2.1667, A 0.000, B 0.000, C 0.000 }
gfCNCPoint2[4432] = {X 517.4752, Y 7.1803, Z -2.1667, A 0.000, B 0.000, C 0.000 }
gfCNCPoint2[4433] = {X 518.2337, Y 6.7038, Z -2.1667, A 0.000, B 0.000, C 0.000 }
gfCNCPoint2[4434] = {X 519.0791, Y 6.4080, Z -2.1667, A 0.000, B 0.000, C 0.000 }
gfCNCPoint2[4435] = {X 519.9692, Y 6.3077, Z -2.1667, A 0.000, B 0.000, C 0.000 }
gfCNCPoint2[4436] = {X 520.6472, Y 6.3079, Z -2.1667, A 0.000, B 0.000, C 0.000 }
gfCNCPoint2[4437] = {X 521.4443, Y 6.3955, Z -2.1667, A 0.000, B 0.000, C 0.000 }
gfCNCPoint2[4438] = {X 522.2079, Y 6.6404, Z -2.1667, A 0.000, B 0.000, C 0.000 }
gfCNCPoint2[4439] = {X 522.9073, Y 7.0327, Z -2.1667, A 0.000, B 0.000, C 0.000 }
gfCNCPoint2[4440] = {X 523.5144, Y 7.5565, Z -2.1667, A 0.000, B 0.000, C 0.000 }
gfCNCPoint2[4441] = {X 524.0048, Y 8.1910, Z -2.1667, A 0.000, B 0.000, C 0.000 }
gfCNCPoint2[4442] = {X 533.9639, Y 8.1913, Z -2.1667, A 0.000, B 0.000, C 0.000 }
gfCNCPoint2[4443] = {X 533.9641, Y 4.1113, Z -2.1667, A 0.000, B 0.000, C 0.000 }
gfCNCPoint2[4444] = {X 533.9641, Y 4.1113, Z 0.8333, A 0.000, B 0.000, C 0.000 }
gfCNCPoint2[4445] = {X 533.9641, Y 4.1113, Z 11.0000, A 0.000, B 0.000, C 0.000 }
gfCNCPoint2[4446] = {X 419.6133, Y 26.5284, Z 11.0000, A 0.000, B 0.000, C 0.000 }
gfCNCPoint2[4447] = {X 419.6133, Y 26.5284, Z 0.8333, A 0.000, B 0.000, C 0.000 }
gfCNCPoint2[4448] = {X 419.6133, Y 26.5284, Z -2.1667, A 0.000, B 0.000, C 0.000 }
gfCNCPoint2[4449] = {X 416.1499, Y 24.3716, Z -2.1667, A 0.000, B 0.000, C 0.000 }
gfCNCPoint2[4450] = {X 411.5460, Y 31.7648, Z -2.1667, A 0.000, B 0.000, C 0.000 }
gfCNCPoint2[4451] = {X 411.5467, Y 40.8984, Z -2.1667, A 0.000, B 0.000, C 0.000 }
gfCNCPoint2[4452] = {X 412.1848, Y 41.5842, Z -2.1667, A 0.000, B 0.000, C 0.000 }
gfCNCPoint2[4453] = {X 412.6650, Y 42.3885, Z -2.1667, A 0.000, B 0.000, C 0.000 }
gfCNCPoint2[4454] = {X 412.9661, Y 43.2755, Z -2.1667, A 0.000, B 0.000, C 0.000 }
gfCNCPoint2[4455] = {X 413.0747, Y 44.2059, Z -2.1667, A 0.000, B 0.000, C 0.000 }
gfCNCPoint2[4456] = {X 413.0747, Y 45.0002, Z -2.1667, A 0.000, B 0.000, C 0.000 }
gfCNCPoint2[4457] = {X 412.9663, Y 45.9614, Z -2.1667, A 0.000, B 0.000, C 0.000 }
gfCNCPoint2[4458] = {X 412.6468, Y 46.8745, Z -2.1667, A 0.000, B 0.000, C 0.000 }
gfCNCPoint2[4459] = {X 412.1321, Y 47.6935, Z -2.1667, A 0.000, B 0.000, C 0.000 }
gfCNCPoint2[4460] = {X 411.4481, Y 48.3776, Z -2.1667, A 0.000, B 0.000, C 0.000 }
gfCNCPoint2[4461] = {X 410.6290, Y 48.8922, Z -2.1667, A 0.000, B 0.000, C 0.000 }
gfCNCPoint2[4462] = {X 409.7159, Y 49.2117, Z -2.1667, A 0.000, B 0.000, C 0.000 }
gfCNCPoint2[4463] = {X 408.7547, Y 49.3200, Z -2.1667, A 0.000, B 0.000, C 0.000 }
gfCNCPoint2[4464] = {X 402.3112, Y 49.3200, Z -2.1667, A 0.000, B 0.000, C 0.000 }
gfCNCPoint2[4465] = {X 401.3546, Y 49.2127, Z -2.1667, A 0.000, B 0.000, C 0.000 }
gfCNCPoint2[4466] = {X 400.4455, Y 48.8963, Z -2.1667, A 0.000, B 0.000, C 0.000 }
gfCNCPoint2[4467] = {X 399.6290, Y 48.3864, Z -2.1667, A 0.000, B 0.000, C 0.000 }
gfCNCPoint2[4468] = {X 398.9457, Y 47.7084, Z -2.1667, A 0.000, B 0.000, C 0.000 }
gfCNCPoint2[4469] = {X 398.4295, Y 46.8959, Z -2.1667, A 0.000, B 0.000, C 0.000 }
gfCNCPoint2[4470] = {X 398.1060, Y 45.9892, Z -2.1667, A 0.000, B 0.000, C 0.000 }
gfCNCPoint2[4471] = {X 397.9913, Y 45.0335, Z -2.1667, A 0.000, B 0.000, C 0.000 }
gfCNCPoint2[4472] = {X 397.9916, Y 44.1528, Z -2.1667, A 0.000, B 0.000, C 0.000 }
gfCNCPoint2[4473] = {X 398.1015, Y 43.2391, Z -2.1667, A 0.000, B 0.000, C 0.000 }
gfCNCPoint2[4474] = {X 398.4024, Y 42.3694, Z -2.1667, A 0.000, B 0.000, C 0.000 }
gfCNCPoint2[4475] = {X 398.8807, Y 41.5832, Z -2.1667, A 0.000, B 0.000, C 0.000 }
gfCNCPoint2[4476] = {X 399.5147, Y 40.9161, Z -2.1667, A 0.000, B 0.000, C 0.000 }
gfCNCPoint2[4477] = {X 399.4729, Y 31.5984, Z -2.1667, A 0.000, B 0.000, C 0.000 }
gfCNCPoint2[4478] = {X 393.3207, Y 20.9004, Z -2.1667, A 0.000, B 0.000, C 0.000 }
gfCNCPoint2[4479] = {X 392.5033, Y 19.5160, Z -2.1667, A 0.000, B 0.000, C 0.000 }
gfCNCPoint2[4480] = {X 391.6541, Y 18.1508, Z -2.1667, A 0.000, B 0.000, C 0.000 }
gfCNCPoint2[4481] = {X 391.1984, Y 17.5271, Z -2.1667, A 0.000, B 0.000, C 0.000 }
gfCNCPoint2[4482] = {X 390.6679, Y 16.9656, Z -2.1667, A 0.000, B 0.000, C 0.000 }
gfCNCPoint2[4483] = {X 389.7909, Y 16.4733, Z -2.1667, A 0.000, B 0.000, C 0.000 }
gfCNCPoint2[4484] = {X 389.0515, Y 15.7916, Z -2.1667, A 0.000, B 0.000, C 0.000 }
gfCNCPoint2[4485] = {X 388.4897, Y 14.9573, Z -2.1667, A 0.000, B 0.000, C 0.000 }
gfCNCPoint2[4486] = {X 388.1361, Y 14.0158, Z -2.1667, A 0.000, B 0.000, C 0.000 }
gfCNCPoint2[4487] = {X 388.0098, Y 13.0180, Z -2.1667, A 0.000, B 0.000, C 0.000 }
gfCNCPoint2[4488] = {X 388.0096, Y 12.1868, Z -2.1667, A 0.000, B 0.000, C 0.000 }
gfCNCPoint2[4489] = {X 388.1179, Y 11.2255, Z -2.1667, A 0.000, B 0.000, C 0.000 }
gfCNCPoint2[4490] = {X 388.4374, Y 10.3125, Z -2.1667, A 0.000, B 0.000, C 0.000 }
gfCNCPoint2[4491] = {X 388.9521, Y 9.4933, Z -2.1667, A 0.000, B 0.000, C 0.000 }
gfCNCPoint2[4492] = {X 389.6361, Y 8.8093, Z -2.1667, A 0.000, B 0.000, C 0.000 }
gfCNCPoint2[4493] = {X 390.4552, Y 8.2946, Z -2.1667, A 0.000, B 0.000, C 0.000 }
gfCNCPoint2[4494] = {X 391.3683, Y 7.9751, Z -2.1667, A 0.000, B 0.000, C 0.000 }
gfCNCPoint2[4495] = {X 392.3296, Y 7.8668, Z -2.1667, A 0.000, B 0.000, C 0.000 }
gfCNCPoint2[4496] = {X 399.1118, Y 7.8668, Z -2.1667, A 0.000, B 0.000, C 0.000 }
gfCNCPoint2[4497] = {X 400.0730, Y 7.9751, Z -2.1667, A 0.000, B 0.000, C 0.000 }
gfCNCPoint2[4498] = {X 400.9861, Y 8.2946, Z -2.1667, A 0.000, B 0.000, C 0.000 }
gfCNCPoint2[4499] = {X 401.8052, Y 8.8093, Z -2.1667, A 0.000, B 0.000, C 0.000 }
gfCNCPoint2[4500] = {X 402.4893, Y 9.4933, Z -2.1667, A 0.000, B 0.000, C 0.000 }
gfCNCPoint2[4501] = {X 403.0039, Y 10.3124, Z -2.1667, A 0.000, B 0.000, C 0.000 }
gfCNCPoint2[4502] = {X 403.3234, Y 11.2255, Z -2.1667, A 0.000, B 0.000, C 0.000 }
gfCNCPoint2[4503] = {X 403.4318, Y 12.1868, Z -2.1667, A 0.000, B 0.000, C 0.000 }
gfCNCPoint2[4504] = {X 403.4318, Y 12.9781, Z -2.1667, A 0.000, B 0.000, C 0.000 }
gfCNCPoint2[4505] = {X 403.3293, Y 13.9134, Z -2.1667, A 0.000, B 0.000, C 0.000 }
gfCNCPoint2[4506] = {X 403.0267, Y 14.8043, Z -2.1667, A 0.000, B 0.000, C 0.000 }
gfCNCPoint2[4507] = {X 405.3571, Y 18.8237, Z -2.1667, A 0.000, B 0.000, C 0.000 }
gfCNCPoint2[4508] = {X 407.8737, Y 14.7545, Z -2.1667, A 0.000, B 0.000, C 0.000 }
gfCNCPoint2[4509] = {X 407.5921, Y 13.9047, Z -2.1667, A 0.000, B 0.000, C 0.000 }
gfCNCPoint2[4510] = {X 407.4917, Y 13.0151, Z -2.1667, A 0.000, B 0.000, C 0.000 }
gfCNCPoint2[4511] = {X 407.4915, Y 12.1868, Z -2.1667, A 0.000, B 0.000, C 0.000 }
gfCNCPoint2[4512] = {X 407.5999, Y 11.2255, Z -2.1667, A 0.000, B 0.000, C 0.000 }
gfCNCPoint2[4513] = {X 407.9194, Y 10.3124, Z -2.1667, A 0.000, B 0.000, C 0.000 }
gfCNCPoint2[4514] = {X 408.4340, Y 9.4933, Z -2.1667, A 0.000, B 0.000, C 0.000 }
gfCNCPoint2[4515] = {X 409.1181, Y 8.8093, Z -2.1667, A 0.000, B 0.000, C 0.000 }
gfCNCPoint2[4516] = {X 409.9372, Y 8.2946, Z -2.1667, A 0.000, B 0.000, C 0.000 }
gfCNCPoint2[4517] = {X 410.8502, Y 7.9751, Z -2.1667, A 0.000, B 0.000, C 0.000 }
gfCNCPoint2[4518] = {X 411.8115, Y 7.8668, Z -2.1667, A 0.000, B 0.000, C 0.000 }
gfCNCPoint2[4519] = {X 419.3245, Y 7.8668, Z -2.1667, A 0.000, B 0.000, C 0.000 }
gfCNCPoint2[4520] = {X 420.2858, Y 7.9751, Z -2.1667, A 0.000, B 0.000, C 0.000 }
gfCNCPoint2[4521] = {X 421.1988, Y 8.2946, Z -2.1667, A 0.000, B 0.000, C 0.000 }
gfCNCPoint2[4522] = {X 422.0179, Y 8.8093, Z -2.1667, A 0.000, B 0.000, C 0.000 }
gfCNCPoint2[4523] = {X 422.7020, Y 9.4933, Z -2.1667, A 0.000, B 0.000, C 0.000 }
gfCNCPoint2[4524] = {X 423.2166, Y 10.3124, Z -2.1667, A 0.000, B 0.000, C 0.000 }
gfCNCPoint2[4525] = {X 423.5361, Y 11.2255, Z -2.1667, A 0.000, B 0.000, C 0.000 }
gfCNCPoint2[4526] = {X 423.6445, Y 12.1868, Z -2.1667, A 0.000, B 0.000, C 0.000 }
gfCNCPoint2[4527] = {X 423.6445, Y 12.9805, Z -2.1667, A 0.000, B 0.000, C 0.000 }
gfCNCPoint2[4528] = {X 423.5510, Y 13.8469, Z -2.1667, A 0.000, B 0.000, C 0.000 }
gfCNCPoint2[4529] = {X 423.2882, Y 14.6778, Z -2.1667, A 0.000, B 0.000, C 0.000 }
gfCNCPoint2[4530] = {X 422.8663, Y 15.4404, Z -2.1667, A 0.000, B 0.000, C 0.000 }
gfCNCPoint2[4531] = {X 422.3020, Y 16.1045, Z -2.1667, A 0.000, B 0.000, C 0.000 }
gfCNCPoint2[4532] = {X 421.6175, Y 16.6440, Z -2.1667, A 0.000, B 0.000, C 0.000 }
gfCNCPoint2[4533] = {X 420.8399, Y 17.0375, Z -2.1667, A 0.000, B 0.000, C 0.000 }
gfCNCPoint2[4534] = {X 420.1236, Y 18.0010, Z -2.1667, A 0.000, B 0.000, C 0.000 }
gfCNCPoint2[4535] = {X 419.4752, Y 19.0115, Z -2.1667, A 0.000, B 0.000, C 0.000 }
gfCNCPoint2[4536] = {X 417.9942, Y 21.4100, Z -2.1667, A 0.000, B 0.000, C 0.000 }
gfCNCPoint2[4537] = {X 416.1499, Y 24.3716, Z -2.1667, A 0.000, B 0.000, C 0.000 }
gfCNCPoint2[4538] = {X 419.5454, Y 26.4861, Z -2.1667, A 0.000, B 0.000, C 0.000 }
gfCNCPoint2[4539] = {X 416.0820, Y 24.3293, Z -2.1667, A 0.000, B 0.000, C 0.000 }
gfCNCPoint2[4540] = {X 411.4660, Y 31.7420, Z -2.1667, A 0.000, B 0.000, C 0.000 }
gfCNCPoint2[4541] = {X 411.4667, Y 40.9350, Z -2.1667, A 0.000, B 0.000, C 0.000 }
gfCNCPoint2[4542] = {X 412.1044, Y 41.6105, Z -2.1667, A 0.000, B 0.000, C 0.000 }
gfCNCPoint2[4543] = {X 412.5847, Y 42.4055, Z -2.1667, A 0.000, B 0.000, C 0.000 }
gfCNCPoint2[4544] = {X 412.8860, Y 43.2842, Z -2.1667, A 0.000, B 0.000, C 0.000 }
gfCNCPoint2[4545] = {X 412.9947, Y 44.2068, Z -2.1667, A 0.000, B 0.000, C 0.000 }
gfCNCPoint2[4546] = {X 412.9947, Y 45.0002, Z -2.1667, A 0.000, B 0.000, C 0.000 }
gfCNCPoint2[4547] = {X 412.8883, Y 45.9436, Z -2.1667, A 0.000, B 0.000, C 0.000 }
gfCNCPoint2[4548] = {X 412.5747, Y 46.8398, Z -2.1667, A 0.000, B 0.000, C 0.000 }
gfCNCPoint2[4549] = {X 412.0696, Y 47.6437, Z -2.1667, A 0.000, B 0.000, C 0.000 }
gfCNCPoint2[4550] = {X 411.3982, Y 48.3150, Z -2.1667, A 0.000, B 0.000, C 0.000 }
gfCNCPoint2[4551] = {X 410.5943, Y 48.8201, Z -2.1667, A 0.000, B 0.000, C 0.000 }
gfCNCPoint2[4552] = {X 409.6981, Y 49.1337, Z -2.1667, A 0.000, B 0.000, C 0.000 }
gfCNCPoint2[4553] = {X 408.7547, Y 49.2400, Z -2.1667, A 0.000, B 0.000, C 0.000 }
gfCNCPoint2[4554] = {X 402.3112, Y 49.2400, Z -2.1667, A 0.000, B 0.000, C 0.000 }
gfCNCPoint2[4555] = {X 401.3723, Y 49.1347, Z -2.1667, A 0.000, B 0.000, C 0.000 }
gfCNCPoint2[4556] = {X 400.4800, Y 48.8242, Z -2.1667, A 0.000, B 0.000, C 0.000 }
gfCNCPoint2[4557] = {X 399.6786, Y 48.3237, Z -2.1667, A 0.000, B 0.000, C 0.000 }
gfCNCPoint2[4558] = {X 399.0080, Y 47.6582, Z -2.1667, A 0.000, B 0.000, C 0.000 }
gfCNCPoint2[4559] = {X 398.5013, Y 46.8608, Z -2.1667, A 0.000, B 0.000, C 0.000 }
gfCNCPoint2[4560] = {X 398.1839, Y 45.9709, Z -2.1667, A 0.000, B 0.000, C 0.000 }
gfCNCPoint2[4561] = {X 398.0713, Y 45.0329, Z -2.1667, A 0.000, B 0.000, C 0.000 }
gfCNCPoint2[4562] = {X 398.0716, Y 44.1538, Z -2.1667, A 0.000, B 0.000, C 0.000 }
gfCNCPoint2[4563] = {X 398.1815, Y 43.2480, Z -2.1667, A 0.000, B 0.000, C 0.000 }
gfCNCPoint2[4564] = {X 398.4827, Y 42.3867, Z -2.1667, A 0.000, B 0.000, C 0.000 }
gfCNCPoint2[4565] = {X 398.9612, Y 41.6098, Z -2.1667, A 0.000, B 0.000, C 0.000 }
gfCNCPoint2[4566] = {X 399.5948, Y 40.9532, Z -2.1667, A 0.000, B 0.000, C 0.000 }
gfCNCPoint2[4567] = {X 399.5528, Y 31.5769, Z -2.1667, A 0.000, B 0.000, C 0.000 }
gfCNCPoint2[4568] = {X 393.3901, Y 20.8605, Z -2.1667, A 0.000, B 0.000, C 0.000 }
gfCNCPoint2[4569] = {X 392.5717, Y 19.4745, Z -2.1667, A 0.000, B 0.000, C 0.000 }
gfCNCPoint2[4570] = {X 391.7216, Y 18.1078, Z -2.1667, A 0.000, B 0.000, C 0.000 }
gfCNCPoint2[4571] = {X 391.2553, Y 17.4703, Z -2.1667, A 0.000, B 0.000, C 0.000 }
gfCNCPoint2[4572] = {X 390.7119, Y 16.8973, Z -2.1667, A 0.000, B 0.000, C 0.000 }
gfCNCPoint2[4573] = {X 389.8472, Y 16.4153, Z -2.1667, A 0.000, B 0.000, C 0.000 }
gfCNCPoint2[4574] = {X 389.1178, Y 15.7460, Z -2.1667, A 0.000, B 0.000, C 0.000 }
gfCNCPoint2[4575] = {X 388.5635, Y 14.9258, Z -2.1667, A 0.000, B 0.000, C 0.000 }
gfCNCPoint2[4576] = {X 388.2145, Y 13.9994, Z -2.1667, A 0.000, B 0.000, C 0.000 }
gfCNCPoint2[4577] = {X 388.0898, Y 13.0173, Z -2.1667, A 0.000, B 0.000, C 0.000 }
gfCNCPoint2[4578] = {X 388.0896, Y 12.1868, Z -2.1667, A 0.000, B 0.000, C 0.000 }
gfCNCPoint2[4579] = {X 388.1959, Y 11.2433, Z -2.1667, A 0.000, B 0.000, C 0.000 }
gfCNCPoint2[4580] = {X 388.5095, Y 10.3472, Z -2.1667, A 0.000, B 0.000, C 0.000 }
gfCNCPoint2[4581] = {X 389.0147, Y 9.5432, Z -2.1667, A 0.000, B 0.000, C 0.000 }
gfCNCPoint2[4582] = {X 389.6860, Y 8.8719, Z -2.1667, A 0.000, B 0.000, C 0.000 }
gfCNCPoint2[4583] = {X 390.4900, Y 8.3667, Z -2.1667, A 0.000, B 0.000, C 0.000 }
gfCNCPoint2[4584] = {X 391.3861, Y 8.0531, Z -2.1667, A 0.000, B 0.000, C 0.000 }
gfCNCPoint2[4585] = {X 392.3296, Y 7.9468, Z -2.1667, A 0.000, B 0.000, C 0.000 }
gfCNCPoint2[4586] = {X 399.1118, Y 7.9468, Z -2.1667, A 0.000, B 0.000, C 0.000 }
gfCNCPoint2[4587] = {X 400.0552, Y 8.0531, Z -2.1667, A 0.000, B 0.000, C 0.000 }
gfCNCPoint2[4588] = {X 400.9514, Y 8.3667, Z -2.1667, A 0.000, B 0.000, C 0.000 }
gfCNCPoint2[4589] = {X 401.7554, Y 8.8718, Z -2.1667, A 0.000, B 0.000, C 0.000 }
gfCNCPoint2[4590] = {X 402.4267, Y 9.5432, Z -2.1667, A 0.000, B 0.000, C 0.000 }
gfCNCPoint2[4591] = {X 402.9319, Y 10.3471, Z -2.1667, A 0.000, B 0.000, C 0.000 }
gfCNCPoint2[4592] = {X 403.2455, Y 11.2433, Z -2.1667, A 0.000, B 0.000, C 0.000 }
gfCNCPoint2[4593] = {X 403.3518, Y 12.1868, Z -2.1667, A 0.000, B 0.000, C 0.000 }
gfCNCPoint2[4594] = {X 403.3518, Y 12.9781, Z -2.1667, A 0.000, B 0.000, C 0.000 }
gfCNCPoint2[4595] = {X 403.2466, Y 13.9164, Z -2.1667, A 0.000, B 0.000, C 0.000 }
gfCNCPoint2[4596] = {X 402.9365, Y 14.8081, Z -2.1667, A 0.000, B 0.000, C 0.000 }
gfCNCPoint2[4597] = {X 405.3549, Y 18.9794, Z -2.1667, A 0.000, B 0.000, C 0.000 }
gfCNCPoint2[4598] = {X 407.9642, Y 14.7601, Z -2.1667, A 0.000, B 0.000, C 0.000 }
gfCNCPoint2[4599] = {X 407.6748, Y 13.9082, Z -2.1667, A 0.000, B 0.000, C 0.000 }
gfCNCPoint2[4600] = {X 407.5717, Y 13.0144, Z -2.1667, A 0.000, B 0.000, C 0.000 }
gfCNCPoint2[4601] = {X 407.5715, Y 12.1868, Z -2.1667, A 0.000, B 0.000, C 0.000 }
gfCNCPoint2[4602] = {X 407.6778, Y 11.2433, Z -2.1667, A 0.000, B 0.000, C 0.000 }
gfCNCPoint2[4603] = {X 407.9914, Y 10.3471, Z -2.1667, A 0.000, B 0.000, C 0.000 }
gfCNCPoint2[4604] = {X 408.4966, Y 9.5432, Z -2.1667, A 0.000, B 0.000, C 0.000 }
gfCNCPoint2[4605] = {X 409.1679, Y 8.8718, Z -2.1667, A 0.000, B 0.000, C 0.000 }
gfCNCPoint2[4606] = {X 409.9719, Y 8.3667, Z -2.1667, A 0.000, B 0.000, C 0.000 }
gfCNCPoint2[4607] = {X 410.8680, Y 8.0531, Z -2.1667, A 0.000, B 0.000, C 0.000 }
gfCNCPoint2[4608] = {X 411.8115, Y 7.9468, Z -2.1667, A 0.000, B 0.000, C 0.000 }
gfCNCPoint2[4609] = {X 419.3245, Y 7.9468, Z -2.1667, A 0.000, B 0.000, C 0.000 }
gfCNCPoint2[4610] = {X 420.2679, Y 8.0531, Z -2.1667, A 0.000, B 0.000, C 0.000 }
gfCNCPoint2[4611] = {X 421.1641, Y 8.3667, Z -2.1667, A 0.000, B 0.000, C 0.000 }
gfCNCPoint2[4612] = {X 421.9681, Y 8.8718, Z -2.1667, A 0.000, B 0.000, C 0.000 }
gfCNCPoint2[4613] = {X 422.6394, Y 9.5432, Z -2.1667, A 0.000, B 0.000, C 0.000 }
gfCNCPoint2[4614] = {X 423.1446, Y 10.3471, Z -2.1667, A 0.000, B 0.000, C 0.000 }
gfCNCPoint2[4615] = {X 423.4582, Y 11.2433, Z -2.1667, A 0.000, B 0.000, C 0.000 }
gfCNCPoint2[4616] = {X 423.5645, Y 12.1868, Z -2.1667, A 0.000, B 0.000, C 0.000 }
gfCNCPoint2[4617] = {X 423.5645, Y 12.9798, Z -2.1667, A 0.000, B 0.000, C 0.000 }
gfCNCPoint2[4618] = {X 423.4720, Y 13.8340, Z -2.1667, A 0.000, B 0.000, C 0.000 }
gfCNCPoint2[4619] = {X 423.2118, Y 14.6528, Z -2.1667, A 0.000, B 0.000, C 0.000 }
gfCNCPoint2[4620] = {X 422.7943, Y 15.4037, Z -2.1667, A 0.000, B 0.000, C 0.000 }
gfCNCPoint2[4621] = {X 422.2361, Y 16.0568, Z -2.1667, A 0.000, B 0.000, C 0.000 }
gfCNCPoint2[4622] = {X 421.5593, Y 16.5861, Z -2.1667, A 0.000, B 0.000, C 0.000 }
gfCNCPoint2[4623] = {X 420.7910, Y 16.9706, Z -2.1667, A 0.000, B 0.000, C 0.000 }
gfCNCPoint2[4624] = {X 420.0642, Y 17.9463, Z -2.1667, A 0.000, B 0.000, C 0.000 }
gfCNCPoint2[4625] = {X 419.4068, Y 18.9701, Z -2.1667, A 0.000, B 0.000, C 0.000 }
gfCNCPoint2[4626] = {X 417.9262, Y 21.3678, Z -2.1667, A 0.000, B 0.000, C 0.000 }
gfCNCPoint2[4627] = {X 416.0820, Y 24.3293, Z -2.1667, A 0.000, B 0.000, C 0.000 }
gfCNCPoint2[4628] = {X 419.4775, Y 26.4438, Z -2.1667, A 0.000, B 0.000, C 0.000 }
gfCNCPoint2[4629] = {X 416.0141, Y 24.2871, Z -2.1667, A 0.000, B 0.000, C 0.000 }
gfCNCPoint2[4630] = {X 411.3860, Y 31.7191, Z -2.1667, A 0.000, B 0.000, C 0.000 }
gfCNCPoint2[4631] = {X 411.3867, Y 40.9721, Z -2.1667, A 0.000, B 0.000, C 0.000 }
gfCNCPoint2[4632] = {X 412.0239, Y 41.6370, Z -2.1667, A 0.000, B 0.000, C 0.000 }
gfCNCPoint2[4633] = {X 412.5044, Y 42.4228, Z -2.1667, A 0.000, B 0.000, C 0.000 }
gfCNCPoint2[4634] = {X 412.8060, Y 43.2930, Z -2.1667, A 0.000, B 0.000, C 0.000 }
gfCNCPoint2[4635] = {X 412.9147, Y 44.2076, Z -2.1667, A 0.000, B 0.000, C 0.000 }
gfCNCPoint2[4636] = {X 412.9147, Y 45.0002, Z -2.1667, A 0.000, B 0.000, C 0.000 }
gfCNCPoint2[4637] = {X 412.8103, Y 45.9258, Z -2.1667, A 0.000, B 0.000, C 0.000 }
gfCNCPoint2[4638] = {X 412.5027, Y 46.8051, Z -2.1667, A 0.000, B 0.000, C 0.000 }
gfCNCPoint2[4639] = {X 412.0070, Y 47.5938, Z -2.1667, A 0.000, B 0.000, C 0.000 }
gfCNCPoint2[4640] = {X 411.3483, Y 48.2525, Z -2.1667, A 0.000, B 0.000, C 0.000 }
gfCNCPoint2[4641] = {X 410.5596, Y 48.7480, Z -2.1667, A 0.000, B 0.000, C 0.000 }
gfCNCPoint2[4642] = {X 409.6803, Y 49.0557, Z -2.1667, A 0.000, B 0.000, C 0.000 }
gfCNCPoint2[4643] = {X 408.7547, Y 49.1600, Z -2.1667, A 0.000, B 0.000, C 0.000 }
gfCNCPoint2[4644] = {X 402.3112, Y 49.1600, Z -2.1667, A 0.000, B 0.000, C 0.000 }
gfCNCPoint2[4645] = {X 401.3900, Y 49.0567, Z -2.1667, A 0.000, B 0.000, C 0.000 }
gfCNCPoint2[4646] = {X 400.5146, Y 48.7520, Z -2.1667, A 0.000, B 0.000, C 0.000 }
gfCNCPoint2[4647] = {X 399.7283, Y 48.2610, Z -2.1667, A 0.000, B 0.000, C 0.000 }
gfCNCPoint2[4648] = {X 399.0703, Y 47.6081, Z -2.1667, A 0.000, B 0.000, C 0.000 }
gfCNCPoint2[4649] = {X 398.5732, Y 46.8257, Z -2.1667, A 0.000, B 0.000, C 0.000 }
gfCNCPoint2[4650] = {X 398.2617, Y 45.9526, Z -2.1667, A 0.000, B 0.000, C 0.000 }
gfCNCPoint2[4651] = {X 398.1513, Y 45.0322, Z -2.1667, A 0.000, B 0.000, C 0.000 }
gfCNCPoint2[4652] = {X 398.1516, Y 44.1549, Z -2.1667, A 0.000, B 0.000, C 0.000 }
gfCNCPoint2[4653] = {X 398.2616, Y 43.2570, Z -2.1667, A 0.000, B 0.000, C 0.000 }
gfCNCPoint2[4654] = {X 398.5630, Y 42.4041, Z -2.1667, A 0.000, B 0.000, C 0.000 }
gfCNCPoint2[4655] = {X 399.0417, Y 41.6366, Z -2.1667, A 0.000, B 0.000, C 0.000 }
gfCNCPoint2[4656] = {X 399.6750, Y 40.9907, Z -2.1667, A 0.000, B 0.000, C 0.000 }
gfCNCPoint2[4657] = {X 399.6327, Y 31.5554, Z -2.1667, A 0.000, B 0.000, C 0.000 }
gfCNCPoint2[4658] = {X 393.4594, Y 20.8206, Z -2.1667, A 0.000, B 0.000, C 0.000 }
gfCNCPoint2[4659] = {X 392.6401, Y 19.4330, Z -2.1667, A 0.000, B 0.000, C 0.000 }
gfCNCPoint2[4660] = {X 391.7890, Y 18.0647, Z -2.1667, A 0.000, B 0.000, C 0.000 }
gfCNCPoint2[4661] = {X 391.3121, Y 17.4135, Z -2.1667, A 0.000, B 0.000, C 0.000 }
gfCNCPoint2[4662] = {X 390.7556, Y 16.8287, Z -2.1667, A 0.000, B 0.000, C 0.000 }
gfCNCPoint2[4663] = {X 389.9033, Y 16.3571, Z -2.1667, A 0.000, B 0.000, C 0.000 }
gfCNCPoint2[4664] = {X 389.1840, Y 15.7002, Z -2.1667, A 0.000, B 0.000, C 0.000 }
gfCNCPoint2[4665] = {X 388.6372, Y 14.8941, Z -2.1667, A 0.000, B 0.000, C 0.000 }
gfCNCPoint2[4666] = {X 388.2928, Y 13.9829, Z -2.1667, A 0.000, B 0.000, C 0.000 }
gfCNCPoint2[4667] = {X 388.1698, Y 13.0166, Z -2.1667, A 0.000, B 0.000, C 0.000 }
gfCNCPoint2[4668] = {X 388.1696, Y 12.1868, Z -2.1667, A 0.000, B 0.000, C 0.000 }
gfCNCPoint2[4669] = {X 388.2739, Y 11.2611, Z -2.1667, A 0.000, B 0.000, C 0.000 }
gfCNCPoint2[4670] = {X 388.5816, Y 10.3819, Z -2.1667, A 0.000, B 0.000, C 0.000 }
gfCNCPoint2[4671] = {X 389.0772, Y 9.5931, Z -2.1667, A 0.000, B 0.000, C 0.000 }
gfCNCPoint2[4672] = {X 389.7359, Y 8.9344, Z -2.1667, A 0.000, B 0.000, C 0.000 }
gfCNCPoint2[4673] = {X 390.5247, Y 8.4388, Z -2.1667, A 0.000, B 0.000, C 0.000 }
gfCNCPoint2[4674] = {X 391.4039, Y 8.1311, Z -2.1667, A 0.000, B 0.000, C 0.000 }
gfCNCPoint2[4675] = {X 392.3296, Y 8.0268, Z -2.1667, A 0.000, B 0.000, C 0.000 }
gfCNCPoint2[4676] = {X 399.1118, Y 8.0268, Z -2.1667, A 0.000, B 0.000, C 0.000 }
gfCNCPoint2[4677] = {X 400.0374, Y 8.1311, Z -2.1667, A 0.000, B 0.000, C 0.000 }
gfCNCPoint2[4678] = {X 400.9167, Y 8.4388, Z -2.1667, A 0.000, B 0.000, C 0.000 }
gfCNCPoint2[4679] = {X 401.7055, Y 8.9344, Z -2.1667, A 0.000, B 0.000, C 0.000 }
gfCNCPoint2[4680] = {X 402.3642, Y 9.5931, Z -2.1667, A 0.000, B 0.000, C 0.000 }
gfCNCPoint2[4681] = {X 402.8598, Y 10.3819, Z -2.1667, A 0.000, B 0.000, C 0.000 }
gfCNCPoint2[4682] = {X 403.1675, Y 11.2611, Z -2.1667, A 0.000, B 0.000, C 0.000 }
gfCNCPoint2[4683] = {X 403.2718, Y 12.1868, Z -2.1667, A 0.000, B 0.000, C 0.000 }
gfCNCPoint2[4684] = {X 403.2718, Y 12.9781, Z -2.1667, A 0.000, B 0.000, C 0.000 }
gfCNCPoint2[4685] = {X 403.1639, Y 13.9192, Z -2.1667, A 0.000, B 0.000, C 0.000 }
gfCNCPoint2[4686] = {X 402.8459, Y 14.8115, Z -2.1667, A 0.000, B 0.000, C 0.000 }
gfCNCPoint2[4687] = {X 405.3526, Y 19.1350, Z -2.1667, A 0.000, B 0.000, C 0.000 }
gfCNCPoint2[4688] = {X 408.0551, Y 14.7654, Z -2.1667, A 0.000, B 0.000, C 0.000 }
gfCNCPoint2[4689] = {X 407.7576, Y 13.9116, Z -2.1667, A 0.000, B 0.000, C 0.000 }
gfCNCPoint2[4690] = {X 407.6517, Y 13.0137, Z -2.1667, A 0.000, B 0.000, C 0.000 }
gfCNCPoint2[4691] = {X 407.6515, Y 12.1868, Z -2.1667, A 0.000, B 0.000, C 0.000 }
gfCNCPoint2[4692] = {X 407.7558, Y 11.2611, Z -2.1667, A 0.000, B 0.000, C 0.000 }
gfCNCPoint2[4693] = {X 408.0635, Y 10.3819, Z -2.1667, A 0.000, B 0.000, C 0.000 }
gfCNCPoint2[4694] = {X 408.5591, Y 9.5931, Z -2.1667, A 0.000, B 0.000, C 0.000 }
gfCNCPoint2[4695] = {X 409.2178, Y 8.9344, Z -2.1667, A 0.000, B 0.000, C 0.000 }
gfCNCPoint2[4696] = {X 410.0066, Y 8.4388, Z -2.1667, A 0.000, B 0.000, C 0.000 }
gfCNCPoint2[4697] = {X 410.8859, Y 8.1311, Z -2.1667, A 0.000, B 0.000, C 0.000 }
gfCNCPoint2[4698] = {X 411.8115, Y 8.0268, Z -2.1667, A 0.000, B 0.000, C 0.000 }
gfCNCPoint2[4699] = {X 419.3245, Y 8.0268, Z -2.1667, A 0.000, B 0.000, C 0.000 }
gfCNCPoint2[4700] = {X 420.2501, Y 8.1311, Z -2.1667, A 0.000, B 0.000, C 0.000 }
gfCNCPoint2[4701] = {X 421.1294, Y 8.4388, Z -2.1667, A 0.000, B 0.000, C 0.000 }
gfCNCPoint2[4702] = {X 421.9182, Y 8.9344, Z -2.1667, A 0.000, B 0.000, C 0.000 }
gfCNCPoint2[4703] = {X 422.5769, Y 9.5931, Z -2.1667, A 0.000, B 0.000, C 0.000 }
gfCNCPoint2[4704] = {X 423.0725, Y 10.3819, Z -2.1667, A 0.000, B 0.000, C 0.000 }
gfCNCPoint2[4705] = {X 423.3802, Y 11.2611, Z -2.1667, A 0.000, B 0.000, C 0.000 }
gfCNCPoint2[4706] = {X 423.4845, Y 12.1868, Z -2.1667, A 0.000, B 0.000, C 0.000 }
gfCNCPoint2[4707] = {X 423.4845, Y 12.9792, Z -2.1667, A 0.000, B 0.000, C 0.000 }
gfCNCPoint2[4708] = {X 423.3930, Y 13.8211, Z -2.1667, A 0.000, B 0.000, C 0.000 }
gfCNCPoint2[4709] = {X 423.1355, Y 14.6278, Z -2.1667, A 0.000, B 0.000, C 0.000 }
gfCNCPoint2[4710] = {X 422.7224, Y 15.3670, Z -2.1667, A 0.000, B 0.000, C 0.000 }
gfCNCPoint2[4711] = {X 422.1703, Y 16.0090, Z -2.1667, A 0.000, B 0.000, C 0.000 }
gfCNCPoint2[4712] = {X 421.5013, Y 16.5281, Z -2.1667, A 0.000, B 0.000, C 0.000 }
gfCNCPoint2[4713] = {X 420.7423, Y 16.9035, Z -2.1667, A 0.000, B 0.000, C 0.000 }
gfCNCPoint2[4714] = {X 420.0049, Y 17.8915, Z -2.1667, A 0.000, B 0.000, C 0.000 }
gfCNCPoint2[4715] = {X 419.3384, Y 18.9286, Z -2.1667, A 0.000, B 0.000, C 0.000 }
gfCNCPoint2[4716] = {X 417.8583, Y 21.3257, Z -2.1667, A 0.000, B 0.000, C 0.000 }
gfCNCPoint2[4717] = {X 416.0141, Y 24.2871, Z -2.1667, A 0.000, B 0.000, C 0.000 }
gfCNCPoint2[4718] = {X 419.4096, Y 26.4015, Z -2.1667, A 0.000, B 0.000, C 0.000 }
gfCNCPoint2[4719] = {X 415.9462, Y 24.2448, Z -2.1667, A 0.000, B 0.000, C 0.000 }
gfCNCPoint2[4720] = {X 411.3060, Y 31.6962, Z -2.1667, A 0.000, B 0.000, C 0.000 }
gfCNCPoint2[4721] = {X 411.3067, Y 41.0096, Z -2.1667, A 0.000, B 0.000, C 0.000 }
gfCNCPoint2[4722] = {X 411.9435, Y 41.6639, Z -2.1667, A 0.000, B 0.000, C 0.000 }
gfCNCPoint2[4723] = {X 412.4241, Y 42.4402, Z -2.1667, A 0.000, B 0.000, C 0.000 }
gfCNCPoint2[4724] = {X 412.7259, Y 43.3019, Z -2.1667, A 0.000, B 0.000, C 0.000 }
gfCNCPoint2[4725] = {X 412.8347, Y 44.2085, Z -2.1667, A 0.000, B 0.000, C 0.000 }
gfCNCPoint2[4726] = {X 412.8347, Y 45.0001, Z -2.1667, A 0.000, B 0.000, C 0.000 }
gfCNCPoint2[4727] = {X 412.7324, Y 45.9080, Z -2.1667, A 0.000, B 0.000, C 0.000 }
gfCNCPoint2[4728] = {X 412.4306, Y 46.7703, Z -2.1667, A 0.000, B 0.000, C 0.000 }
gfCNCPoint2[4729] = {X 411.9445, Y 47.5439, Z -2.1667, A 0.000, B 0.000, C 0.000 }
gfCNCPoint2[4730] = {X 411.2985, Y 48.1899, Z -2.1667, A 0.000, B 0.000, C 0.000 }
gfCNCPoint2[4731] = {X 410.5249, Y 48.6760, Z -2.1667, A 0.000, B 0.000, C 0.000 }
gfCNCPoint2[4732] = {X 409.6625, Y 48.9777, Z -2.1667, A 0.000, B 0.000, C 0.000 }
gfCNCPoint2[4733] = {X 408.7547, Y 49.0800, Z -2.1667, A 0.000, B 0.000, C 0.000 }
gfCNCPoint2[4734] = {X 402.3112, Y 49.0800, Z -2.1667, A 0.000, B 0.000, C 0.000 }
gfCNCPoint2[4735] = {X 401.4077, Y 48.9787, Z -2.1667, A 0.000, B 0.000, C 0.000 }
gfCNCPoint2[4736] = {X 400.5491, Y 48.6799, Z -2.1667, A 0.000, B 0.000, C 0.000 }
gfCNCPoint2[4737] = {X 399.7780, Y 48.1983, Z -2.1667, A 0.000, B 0.000, C 0.000 }
gfCNCPoint2[4738] = {X 399.1326, Y 47.5579, Z -2.1667, A 0.000, B 0.000, C 0.000 }
gfCNCPoint2[4739] = {X 398.6451, Y 46.7906, Z -2.1667, A 0.000, B 0.000, C 0.000 }
gfCNCPoint2[4740] = {X 398.3396, Y 45.9343, Z -2.1667, A 0.000, B 0.000, C 0.000 }
gfCNCPoint2[4741] = {X 398.2313, Y 45.0316, Z -2.1667, A 0.000, B 0.000, C 0.000 }
gfCNCPoint2[4742] = {X 398.2316, Y 44.1559, Z -2.1667, A 0.000, B 0.000, C 0.000 }
gfCNCPoint2[4743] = {X 398.3416, Y 43.2661, Z -2.1667, A 0.000, B 0.000, C 0.000 }
gfCNCPoint2[4744] = {X 398.6434, Y 42.4218, Z -2.1667, A 0.000, B 0.000, C 0.000 }
gfCNCPoint2[4745] = {X 399.1223, Y 41.6638, Z -2.1667, A 0.000, B 0.000, C 0.000 }
gfCNCPoint2[4746] = {X 399.7552, Y 41.0287, Z -2.1667, A 0.000, B 0.000, C 0.000 }
gfCNCPoint2[4747] = {X 399.7126, Y 31.5338, Z -2.1667, A 0.000, B 0.000, C 0.000 }
gfCNCPoint2[4748] = {X 393.5288, Y 20.7807, Z -2.1667, A 0.000, B 0.000, C 0.000 }
gfCNCPoint2[4749] = {X 392.7085, Y 19.3916, Z -2.1667, A 0.000, B 0.000, C 0.000 }
gfCNCPoint2[4750] = {X 391.8565, Y 18.0217, Z -2.1667, A 0.000, B 0.000, C 0.000 }
gfCNCPoint2[4751] = {X 391.3688, Y 17.3566, Z -2.1667, A 0.000, B 0.000, C 0.000 }
gfCNCPoint2[4752] = {X 390.7992, Y 16.7601, Z -2.1667, A 0.000, B 0.000, C 0.000 }
gfCNCPoint2[4753] = {X 389.9593, Y 16.2988, Z -2.1667, A 0.000, B 0.000, C 0.000 }
gfCNCPoint2[4754] = {X 389.2501, Y 15.6544, Z -2.1667, A 0.000, B 0.000, C 0.000 }
gfCNCPoint2[4755] = {X 388.7108, Y 14.8623, Z -2.1667, A 0.000, B 0.000, C 0.000 }
gfCNCPoint2[4756] = {X 388.3711, Y 13.9663, Z -2.1667, A 0.000, B 0.000, C 0.000 }
gfCNCPoint2[4757] = {X 388.2498, Y 13.0158, Z -2.1667, A 0.000, B 0.000, C 0.000 }
gfCNCPoint2[4758] = {X 388.2496, Y 12.1868, Z -2.1667, A 0.000, B 0.000, C 0.000 }
gfCNCPoint2[4759] = {X 388.3519, Y 11.2789, Z -2.1667, A 0.000, B 0.000, C 0.000 }
gfCNCPoint2[4760] = {X 388.6537, Y 10.4166, Z -2.1667, A 0.000, B 0.000, C 0.000 }
gfCNCPoint2[4761] = {X 389.1398, Y 9.6430, Z -2.1667, A 0.000, B 0.000, C 0.000 }
gfCNCPoint2[4762] = {X 389.7858, Y 8.9969, Z -2.1667, A 0.000, B 0.000, C 0.000 }
gfCNCPoint2[4763] = {X 390.5594, Y 8.5109, Z -2.1667, A 0.000, B 0.000, C 0.000 }
gfCNCPoint2[4764] = {X 391.4217, Y 8.2091, Z -2.1667, A 0.000, B 0.000, C 0.000 }
gfCNCPoint2[4765] = {X 392.3296, Y 8.1068, Z -2.1667, A 0.000, B 0.000, C 0.000 }
gfCNCPoint2[4766] = {X 399.1118, Y 8.1068, Z -2.1667, A 0.000, B 0.000, C 0.000 }
gfCNCPoint2[4767] = {X 400.0196, Y 8.2091, Z -2.1667, A 0.000, B 0.000, C 0.000 }
gfCNCPoint2[4768] = {X 400.8820, Y 8.5109, Z -2.1667, A 0.000, B 0.000, C 0.000 }
gfCNCPoint2[4769] = {X 401.6556, Y 8.9969, Z -2.1667, A 0.000, B 0.000, C 0.000 }
gfCNCPoint2[4770] = {X 402.3016, Y 9.6430, Z -2.1667, A 0.000, B 0.000, C 0.000 }
gfCNCPoint2[4771] = {X 402.7877, Y 10.4166, Z -2.1667, A 0.000, B 0.000, C 0.000 }
gfCNCPoint2[4772] = {X 403.0895, Y 11.2789, Z -2.1667, A 0.000, B 0.000, C 0.000 }
gfCNCPoint2[4773] = {X 403.1918, Y 12.1868, Z -2.1667, A 0.000, B 0.000, C 0.000 }
gfCNCPoint2[4774] = {X 403.1918, Y 12.9781, Z -2.1667, A 0.000, B 0.000, C 0.000 }
gfCNCPoint2[4775] = {X 403.0811, Y 13.9218, Z -2.1667, A 0.000, B 0.000, C 0.000 }
gfCNCPoint2[4776] = {X 402.7551, Y 14.8144, Z -2.1667, A 0.000, B 0.000, C 0.000 }
gfCNCPoint2[4777] = {X 405.3504, Y 19.2907, Z -2.1667, A 0.000, B 0.000, C 0.000 }
gfCNCPoint2[4778] = {X 408.1462, Y 14.7701, Z -2.1667, A 0.000, B 0.000, C 0.000 }
gfCNCPoint2[4779] = {X 408.1095, Y 14.6931, Z -2.1667, A 0.000, B 0.000, C 0.000 }
gfCNCPoint2[4780] = {X 408.0745, Y 14.6153, Z -2.1667, A 0.000, B 0.000, C 0.000 }
gfCNCPoint2[4781] = {X 407.8218, Y 13.8316, Z -2.1667, A 0.000, B 0.000, C 0.000 }
gfCNCPoint2[4782] = {X 407.7317, Y 13.0131, Z -2.1667, A 0.000, B 0.000, C 0.000 }
gfCNCPoint2[4783] = {X 407.7315, Y 12.1868, Z -2.1667, A 0.000, B 0.000, C 0.000 }
gfCNCPoint2[4784] = {X 407.8338, Y 11.2789, Z -2.1667, A 0.000, B 0.000, C 0.000 }
gfCNCPoint2[4785] = {X 408.1356, Y 10.4166, Z -2.1667, A 0.000, B 0.000, C 0.000 }
gfCNCPoint2[4786] = {X 408.6217, Y 9.6430, Z -2.1667, A 0.000, B 0.000, C 0.000 }
gfCNCPoint2[4787] = {X 409.2677, Y 8.9969, Z -2.1667, A 0.000, B 0.000, C 0.000 }
gfCNCPoint2[4788] = {X 410.0413, Y 8.5109, Z -2.1667, A 0.000, B 0.000, C 0.000 }
gfCNCPoint2[4789] = {X 410.9037, Y 8.2091, Z -2.1667, A 0.000, B 0.000, C 0.000 }
gfCNCPoint2[4790] = {X 411.8115, Y 8.1068, Z -2.1667, A 0.000, B 0.000, C 0.000 }
gfCNCPoint2[4791] = {X 419.3245, Y 8.1068, Z -2.1667, A 0.000, B 0.000, C 0.000 }
gfCNCPoint2[4792] = {X 420.2323, Y 8.2091, Z -2.1667, A 0.000, B 0.000, C 0.000 }
gfCNCPoint2[4793] = {X 421.0947, Y 8.5109, Z -2.1667, A 0.000, B 0.000, C 0.000 }
gfCNCPoint2[4794] = {X 421.8683, Y 8.9969, Z -2.1667, A 0.000, B 0.000, C 0.000 }
gfCNCPoint2[4795] = {X 422.5143, Y 9.6430, Z -2.1667, A 0.000, B 0.000, C 0.000 }
gfCNCPoint2[4796] = {X 423.0004, Y 10.4166, Z -2.1667, A 0.000, B 0.000, C 0.000 }
gfCNCPoint2[4797] = {X 423.3022, Y 11.2789, Z -2.1667, A 0.000, B 0.000, C 0.000 }
gfCNCPoint2[4798] = {X 423.4045, Y 12.1868, Z -2.1667, A 0.000, B 0.000, C 0.000 }
gfCNCPoint2[4799] = {X 423.4045, Y 12.9786, Z -2.1667, A 0.000, B 0.000, C 0.000 }
gfCNCPoint2[4800] = {X 423.3139, Y 13.8080, Z -2.1667, A 0.000, B 0.000, C 0.000 }
gfCNCPoint2[4801] = {X 423.0592, Y 14.6026, Z -2.1667, A 0.000, B 0.000, C 0.000 }
gfCNCPoint2[4802] = {X 422.6506, Y 15.3301, Z -2.1667, A 0.000, B 0.000, C 0.000 }
gfCNCPoint2[4803] = {X 422.1046, Y 15.9611, Z -2.1667, A 0.000, B 0.000, C 0.000 }
gfCNCPoint2[4804] = {X 421.4434, Y 16.4700, Z -2.1667, A 0.000, B 0.000, C 0.000 }
gfCNCPoint2[4805] = {X 420.6937, Y 16.8362, Z -2.1667, A 0.000, B 0.000, C 0.000 }
gfCNCPoint2[4806] = {X 419.9456, Y 17.8366, Z -2.1667, A 0.000, B 0.000, C 0.000 }
gfCNCPoint2[4807] = {X 419.2699, Y 18.8871, Z -2.1667, A 0.000, B 0.000, C 0.000 }
gfCNCPoint2[4808] = {X 417.7903, Y 21.2835, Z -2.1667, A 0.000, B 0.000, C 0.000 }
gfCNCPoint2[4809] = {X 415.9462, Y 24.2448, Z -2.1667, A 0.000, B 0.000, C 0.000 }
gfCNCPoint2[4810] = {X 419.3417, Y 26.3592, Z -2.1667, A 0.000, B 0.000, C 0.000 }
gfCNCPoint2[4811] = {X 415.8783, Y 24.2025, Z -2.1667, A 0.000, B 0.000, C 0.000 }
gfCNCPoint2[4812] = {X 411.2260, Y 31.6734, Z -2.1667, A 0.000, B 0.000, C 0.000 }
gfCNCPoint2[4813] = {X 411.2267, Y 41.0475, Z -2.1667, A 0.000, B 0.000, C 0.000 }
gfCNCPoint2[4814] = {X 411.8630, Y 41.6909, Z -2.1667, A 0.000, B 0.000, C 0.000 }
gfCNCPoint2[4815] = {X 412.3437, Y 42.4576, Z -2.1667, A 0.000, B 0.000, C 0.000 }
gfCNCPoint2[4816] = {X 412.6458, Y 43.3106, Z -2.1667, A 0.000, B 0.000, C 0.000 }
gfCNCPoint2[4817] = {X 412.7547, Y 44.2089, Z -2.1667, A 0.000, B 0.000, C 0.000 }
gfCNCPoint2[4818] = {X 412.7545, Y 45.0384, Z -2.1667, A 0.000, B 0.000, C 0.000 }
gfCNCPoint2[4819] = {X 412.6469, Y 45.9222, Z -2.1667, A 0.000, B 0.000, C 0.000 }
gfCNCPoint2[4820] = {X 412.3466, Y 46.7602, Z -2.1667, A 0.000, B 0.000, C 0.000 }
gfCNCPoint2[4821] = {X 411.8683, Y 47.5111, Z -2.1667, A 0.000, B 0.000, C 0.000 }
gfCNCPoint2[4822] = {X 411.2357, Y 48.1376, Z -2.1667, A 0.000, B 0.000, C 0.000 }
gfCNCPoint2[4823] = {X 410.4803, Y 48.6086, Z -2.1667, A 0.000, B 0.000, C 0.000 }
gfCNCPoint2[4824] = {X 409.6394, Y 48.9009, Z -2.1667, A 0.000, B 0.000, C 0.000 }
gfCNCPoint2[4825] = {X 408.7547, Y 49.0000, Z -2.1667, A 0.000, B 0.000, C 0.000 }
gfCNCPoint2[4826] = {X 402.3112, Y 49.0000, Z -2.1667, A 0.000, B 0.000, C 0.000 }
gfCNCPoint2[4827] = {X 401.4211, Y 48.8997, Z -2.1667, A 0.000, B 0.000, C 0.000 }
gfCNCPoint2[4828] = {X 400.5757, Y 48.6039, Z -2.1667, A 0.000, B 0.000, C 0.000 }
gfCNCPoint2[4829] = {X 399.8172, Y 48.1273, Z -2.1667, A 0.000, B 0.000, C 0.000 }
gfCNCPoint2[4830] = {X 399.1839, Y 47.4939, Z -2.1667, A 0.000, B 0.000, C 0.000 }
gfCNCPoint2[4831] = {X 398.7073, Y 46.7355, Z -2.1667, A 0.000, B 0.000, C 0.000 }
gfCNCPoint2[4832] = {X 398.4115, Y 45.8900, Z -2.1667, A 0.000, B 0.000, C 0.000 }
gfCNCPoint2[4833] = {X 398.3112, Y 45.0000, Z -2.1667, A 0.000, B 0.000, C 0.000 }
gfCNCPoint2[4834] = {X 398.3115, Y 44.1569, Z -2.1667, A 0.000, B 0.000, C 0.000 }
